LIN {X 0,Y 376.108,Z 924.328,A -85,B 0,C 180,E1 13646.479,E2 13646.479} C_VEL
LIN {X 0,Y 367.775,Z 908.146,A -85,B 0,C 180,E1 13649.429,E2 13649.429} C_VEL
LIN {X 0,Y 364.4,Z 915.516,A -85,B 0,C 180,E1 13649.758,E2 13649.758} C_VEL
LIN {X 0,Y 357.895,Z 928.85,A -85,B 0,C 180,E1 13650.369,E2 13650.369} C_VEL
LIN {X 0,Y 353.873,Z 934.95,A -85,B 0,C 180,E1 13650.878,E2 13650.878} C_VEL
LIN {X 0,Y 348.654,Z 943.219,A -85,B 0,C 180,E1 13651.467,E2 13651.467} C_VEL
LIN {X 0,Y 345.906,Z 946.107,A -85,B 0,C 180,E1 13652.021,E2 13652.021} C_VEL
LIN {X 0,Y 343.36,Z 977.029,A -85,B 0,C 180,E1 13654.434,E2 13654.434} C_VEL
LIN {X 0,Y 340.02,Z 1003.082,A -85,B 0,C 180,E1 13657.588,E2 13657.588} C_VEL
LIN {X 0,Y 336.523,Z 1024.234,A -85,B 0,C 180,E1 13661.411,E2 13661.411} C_VEL
LIN {X 0,Y 333.51,Z 1039.452,A -85,B 0,C 180,E1 13665.541,E2 13665.541} C_VEL
LIN {X 0,Y 331.006,Z 1050.175,A -85,B 0,C 180,E1 13670.2,E2 13670.2} C_VEL
LIN {X 0,Y 329.716,Z 1055.388,A -85,B 0,C 180,E1 13674.73,E2 13674.73} C_VEL
LIN {X 0,Y 328.873,Z 1055.973,A -85,B 0,C 180,E1 13679.999,E2 13679.999} C_VEL
LIN {X 0,Y 328.837,Z 1050.81,A -85,B 0,C 180,E1 13685.282,E2 13685.282} C_VEL
LIN {X 0,Y 329.705,Z 1039.548,A -85,B 0,C 180,E1 13690.582,E2 13690.582} C_VEL
LIN {X 0,Y 331.439,Z 1023.575,A -85,B 0,C 180,E1 13695.226,E2 13695.226} C_VEL
LIN {X 0,Y 334.022,Z 1001.735,A -85,B 0,C 180,E1 13699.527,E2 13699.527} C_VEL
LIN {X 0,Y 337.182,Z 974.565,A -85,B 0,C 180,E1 13703.187,E2 13703.187} C_VEL
LIN {X 0,Y 339.904,Z 944.159,A -85,B 0,C 180,E1 13705.915,E2 13705.915} C_VEL
LIN {X 0,Y 341.977,Z 913.832,A -85,B 0,C 180,E1 13707.697,E2 13707.697} C_VEL
LIN {X 0,Y 345.152,Z 909.514,A -85,B 0,C 180,E1 13708.423,E2 13708.423} C_VEL
LIN {X 0,Y 349.954,Z 896.791,A -85,B 0,C 180,E1 13709.156,E2 13709.156} C_VEL
LIN {X 0,Y 354.172,Z 888.97,A -85,B 0,C 180,E1 13710.083,E2 13710.083} C_VEL
LIN {X 0,Y 355.518,Z 886.512,A -85,B 0,C 180,E1 13710.372,E2 13710.372} C_VEL
LIN {X 0,Y 370.198,Z 910.648,A -85,B 0,C 180,E1 13715.495,E2 13715.495} C_VEL
LIN {X 0,Y 383.568,Z 939.518,A -85,B 0,C 180,E1 13720.262,E2 13720.262} C_VEL
LIN {X 0,Y 386.458,Z 948.208,A -85,B 0,C 180,E1 13721.491,E2 13721.491} C_VEL
LIN {X 0,Y 378.77,Z 984.053,A -85,B 0,C 180,E1 13723.63,E2 13723.63} C_VEL
LIN {X 0,Y 369.066,Z 1018.522,A -85,B 0,C 180,E1 13726.591,E2 13726.591} C_VEL
LIN {X 0,Y 358.745,Z 1049.661,A -85,B 0,C 180,E1 13730.368,E2 13730.368} C_VEL
LIN {X 0,Y 348.828,Z 1076.763,A -85,B 0,C 180,E1 13734.89,E2 13734.89} C_VEL
LIN {X 0,Y 339.261,Z 1101.55,A -85,B 0,C 180,E1 13740.597,E2 13740.597} C_VEL
LIN {X 0,Y 332.687,Z 1119.974,A -85,B 0,C 180,E1 13746.531,E2 13746.531} C_VEL
LIN {X 0,Y 328.362,Z 1134.473,A -85,B 0,C 180,E1 13753.249,E2 13753.249} C_VEL
LIN {X 0,Y 326.282,Z 1144.274,A -85,B 0,C 180,E1 13760.651,E2 13760.651} C_VEL
LIN {X 0,Y 325.694,Z 1148.277,A -85,B 0,C 180,E1 13767.334,E2 13767.334} C_VEL
LIN {X 0,Y 325.744,Z 1148.241,A -85,B 0,C 180,E1 13772.663,E2 13772.663} C_VEL
LIN {X 0,Y 326.287,Z 1144.195,A -85,B 0,C 180,E1 13779.346,E2 13779.346} C_VEL
LIN {X 0,Y 328.377,Z 1134.321,A -85,B 0,C 180,E1 13786.748,E2 13786.748} C_VEL
LIN {X 0,Y 332.774,Z 1119.754,A -85,B 0,C 180,E1 13793.46,E2 13793.46} C_VEL
LIN {X 0,Y 340.29,Z 1099.046,A -85,B 0,C 180,E1 13799.987,E2 13799.987} C_VEL
LIN {X 0,Y 350.198,Z 1073.11,A -85,B 0,C 180,E1 13805.709,E2 13805.709} C_VEL
LIN {X 0,Y 360.949,Z 1043.194,A -85,B 0,C 180,E1 13810.431,E2 13810.431} C_VEL
LIN {X 0,Y 371.664,Z 1010.049,A -85,B 0,C 180,E1 13814.133,E2 13814.133} C_VEL
LIN {X 0,Y 381.081,Z 973.71,A -85,B 0,C 180,E1 13816.999,E2 13816.999} C_VEL
LIN {X 0,Y 386.353,Z 946.977,A -85,B 0,C 180,E1 13818.517,E2 13818.517} C_VEL
LIN {X 0,Y 374.373,Z 918.78,A -85,B 0,C 180,E1 13822.931,E2 13822.931} C_VEL
LIN {X 0,Y 360.213,Z 893.932,A -85,B 0,C 180,E1 13827.801,E2 13827.801} C_VEL
LIN {X 0,Y 347.294,Z 875.046,A -85,B 0,C 180,E1 13832.671,E2 13832.671} C_VEL
LIN {X 0,Y 339.642,Z 864.701,A -85,B 0,C 180,E1 13836.146,E2 13836.146} C_VEL
LIN {X 0,Y 334.753,Z 857.931,A -85,B 0,C 180,E1 13838.79,E2 13838.79} C_VEL
LIN {X 0,Y 330.751,Z 852.629,A -85,B 0,C 180,E1 13841.314,E2 13841.314} C_VEL
LIN {X 0,Y 329.425,Z 850.767,A -85,B 0,C 180,E1 13842.257,E2 13842.257} C_VEL
LIN {X 0,Y 325.061,Z 845.874,A -85,B 0,C 180,E1 13845.848,E2 13845.848} C_VEL
LIN {X 0,Y 324.743,Z 843.44,A -85,B 0,C 180,E1 13846.522,E2 13846.522} C_VEL
LIN {X 0,Y 325.226,Z 843.44,A -85,B 0,C 180,E1 13854.659,E2 13854.659} C_VEL
LIN {X 0,Y 325.59,Z 843.44,A -85,B 0,C 180,E1 13860.001,E2 13860.001} C_VEL
LIN {X 0,Y 324.995,Z 843.44,A -85,B 0,C 180,E1 13868.035,E2 13868.035} C_VEL
LIN {X 0,Y 324.861,Z 844.009,A -85,B 0,C 180,E1 13869.304,E2 13869.304} C_VEL
LIN {X 0,Y 327.183,Z 849.216,A -85,B 0,C 180,E1 13871.617,E2 13871.617} C_VEL
LIN {X 0,Y 330.663,Z 851.939,A -85,B 0,C 180,E1 13874.079,E2 13874.079} C_VEL
LIN {X 0,Y 334.613,Z 857.811,A -85,B 0,C 180,E1 13876.641,E2 13876.641} C_VEL
LIN {X 0,Y 336.707,Z 860.625,A -85,B 0,C 180,E1 13877.835,E2 13877.835} C_VEL
LIN {X 0,Y 342.23,Z 868.171,A -85,B 0,C 180,E1 13880.646,E2 13880.646} C_VEL
LIN {X 0,Y 351.334,Z 880.835,A -85,B 0,C 180,E1 13884.527,E2 13884.527} C_VEL
LIN {X 0,Y 365.006,Z 902.571,A -85,B 0,C 180,E1 13889.594,E2 13889.594} C_VEL
LIN {X 0,Y 378.204,Z 929.229,A -85,B 0,C 180,E1 13894.346,E2 13894.346} C_VEL
LIN {X 0,Y 385.902,Z 951.03,A -85,B 0,C 180,E1 13897.51,E2 13897.51} C_VEL
LIN {X 0,Y 376.987,Z 993.57,A -85,B 0,C 180,E1 13900.262,E2 13900.262} C_VEL
LIN {X 0,Y 366.594,Z 1031.143,A -85,B 0,C 180,E1 13903.716,E2 13903.716} C_VEL
LIN {X 0,Y 355.486,Z 1065.912,A -85,B 0,C 180,E1 13908.156,E2 13908.156} C_VEL
LIN {X 0,Y 344.895,Z 1097.163,A -85,B 0,C 180,E1 13913.655,E2 13913.655} C_VEL
LIN {X 0,Y 336.481,Z 1122.605,A -85,B 0,C 180,E1 13919.764,E2 13919.764} C_VEL
LIN {X 0,Y 330.265,Z 1143.966,A -85,B 0,C 180,E1 13926.842,E2 13926.842} C_VEL
LIN {X 0,Y 327.114,Z 1158.659,A -85,B 0,C 180,E1 13933.877,E2 13933.877} C_VEL
LIN {X 0,Y 325.913,Z 1167.658,A -85,B 0,C 180,E1 13940.643,E2 13940.643} C_VEL
LIN {X 0,Y 325.706,Z 1171.943,A -85,B 0,C 180,E1 13947.337,E2 13947.337} C_VEL
LIN {X 0,Y 325.641,Z 1171.94,A -85,B 0,C 180,E1 13952.666,E2 13952.666} C_VEL
LIN {X 0,Y 325.91,Z 1167.658,A -85,B 0,C 180,E1 13959.359,E2 13959.359} C_VEL
LIN {X 0,Y 327.121,Z 1158.659,A -85,B 0,C 180,E1 13966.125,E2 13966.125} C_VEL
LIN {X 0,Y 330.278,Z 1143.971,A -85,B 0,C 180,E1 13973.159,E2 13973.159} C_VEL
LIN {X 0,Y 336.415,Z 1122.636,A -85,B 0,C 180,E1 13980.237,E2 13980.237} C_VEL
LIN {X 0,Y 338.564,Z 1116.059,A -85,B 0,C 180,E1 13981.992,E2 13981.992} C_VEL
LIN {X 0,Y 338.171,Z 1107.045,A -85,B 0,C 180,E1 13984.532,E2 13984.532} C_VEL
LIN {X 0,Y 338.05,Z 1097.476,A -85,B 0,C 180,E1 13987.029,E2 13987.029} C_VEL
LIN {X 0,Y 349.215,Z 1066.113,A -85,B 0,C 180,E1 13992.655,E2 13992.655} C_VEL
LIN {X 0,Y 361.147,Z 1029.977,A -85,B 0,C 180,E1 13997.312,E2 13997.312} C_VEL
LIN {X 0,Y 372.132,Z 991.554,A -85,B 0,C 180,E1 14000.812,E2 14000.812} C_VEL
LIN {X 0,Y 380.39,Z 954.941,A -85,B 0,C 180,E1 14003.166,E2 14003.166} C_VEL
LIN {X 0,Y 371.021,Z 928.372,A -85,B 0,C 180,E1 14007.27,E2 14007.27} C_VEL
LIN {X 0,Y 366.968,Z 920.536,A -85,B 0,C 180,E1 14008.782,E2 14008.782} C_VEL
LIN {X 0,Y 359.568,Z 934.219,A -85,B 0,C 180,E1 14009.476,E2 14009.476} C_VEL
LIN {X 0,Y 350.055,Z 948.399,A -85,B 0,C 180,E1 14010.519,E2 14010.519} C_VEL
LIN {X 0,Y 340.44,Z 959.968,A -85,B 0,C 180,E1 14011.802,E2 14011.802} C_VEL
LIN {X 0,Y 338.533,Z 961.854,A -85,B 0,C 180,E1 14012.264,E2 14012.264} C_VEL
LIN {X 0,Y 335.38,Z 990.271,A -85,B 0,C 180,E1 14015.018,E2 14015.018} C_VEL
LIN {X 0,Y 331.905,Z 1012.677,A -85,B 0,C 180,E1 14018.245,E2 14018.245} C_VEL
LIN {X 0,Y 328.372,Z 1031.449,A -85,B 0,C 180,E1 14022.214,E2 14022.214} C_VEL
LIN {X 0,Y 325.27,Z 1045.038,A -85,B 0,C 180,E1 14026.541,E2 14026.541} C_VEL
LIN {X 0,Y 323.081,Z 1053.423,A -85,B 0,C 180,E1 14030.93,E2 14030.93} C_VEL
LIN {X 0,Y 322.031,Z 1057.041,A -85,B 0,C 180,E1 14034.604,E2 14034.604} C_VEL
LIN {X 0,Y 321.112,Z 1057.42,A -85,B 0,C 180,E1 14039.999,E2 14039.999} C_VEL
LIN {X 0,Y 321.084,Z 1052.008,A -85,B 0,C 180,E1 14045.41,E2 14045.41} C_VEL
LIN {X 0,Y 321.743,Z 1042.227,A -85,B 0,C 180,E1 14050.161,E2 14050.161} C_VEL
LIN {X 0,Y 323.495,Z 1026.843,A -85,B 0,C 180,E1 14054.914,E2 14054.914} C_VEL
LIN {X 0,Y 326.047,Z 1005.884,A -85,B 0,C 180,E1 14059.318,E2 14059.318} C_VEL
LIN {X 0,Y 329.216,Z 979.656,A -85,B 0,C 180,E1 14063.094,E2 14063.094} C_VEL
LIN {X 0,Y 332.106,Z 949.359,A -85,B 0,C 180,E1 14066.024,E2 14066.024} C_VEL
LIN {X 0,Y 333.389,Z 936.954,A -85,B 0,C 180,E1 14067.006,E2 14067.006} C_VEL
LIN {X 0,Y 337.196,Z 932.766,A -85,B 0,C 180,E1 14067.905,E2 14067.905} C_VEL
LIN {X 0,Y 344.097,Z 918.915,A -85,B 0,C 180,E1 14068.872,E2 14068.872} C_VEL
LIN {X 0,Y 349.104,Z 909.69,A -85,B 0,C 180,E1 14069.726,E2 14069.726} C_VEL
LIN {X 0,Y 352.399,Z 901.513,A -85,B 0,C 180,E1 14070.21,E2 14070.21} C_VEL
LIN {X 0,Y 355.375,Z 897.164,A -85,B 0,C 180,E1 14070.839,E2 14070.839} C_VEL
LIN {X 0,Y 369.602,Z 923.178,A -85,B 0,C 180,E1 14076.163,E2 14076.163} C_VEL
LIN {X 0,Y 380.719,Z 949.941,A -85,B 0,C 180,E1 14080.564,E2 14080.564} C_VEL
LIN {X 0,Y 372.121,Z 989.556,A -85,B 0,C 180,E1 14083.105,E2 14083.105} C_VEL
LIN {X 0,Y 361.673,Z 1024.445,A -85,B 0,C 180,E1 14086.308,E2 14086.308} C_VEL
LIN {X 0,Y 349.978,Z 1057.121,A -85,B 0,C 180,E1 14090.582,E2 14090.582} C_VEL
LIN {X 0,Y 339.324,Z 1084.484,A -85,B 0,C 180,E1 14095.629,E2 14095.629} C_VEL
LIN {X 0,Y 330.036,Z 1107.705,A -85,B 0,C 180,E1 14101.615,E2 14101.615} C_VEL
LIN {X 0,Y 323.268,Z 1126.436,A -85,B 0,C 180,E1 14108.571,E2 14108.571} C_VEL
LIN {X 0,Y 319.816,Z 1138.047,A -85,B 0,C 180,E1 14114.905,E2 14114.905} C_VEL
LIN {X 0,Y 318.195,Z 1145.708,A -85,B 0,C 180,E1 14121.791,E2 14121.791} C_VEL
LIN {X 0,Y 317.815,Z 1148.564,A -85,B 0,C 180,E1 14127.268,E2 14127.268} C_VEL
LIN {X 0,Y 317.845,Z 1148.53,A -85,B 0,C 180,E1 14132.729,E2 14132.729} C_VEL
LIN {X 0,Y 318.441,Z 1144.488,A -85,B 0,C 180,E1 14139.578,E2 14139.578} C_VEL
LIN {X 0,Y 320.716,Z 1134.625,A -85,B 0,C 180,E1 14147.16,E2 14147.16} C_VEL
LIN {X 0,Y 325.391,Z 1120.071,A -85,B 0,C 180,E1 14154.025,E2 14154.025} C_VEL
LIN {X 0,Y 333.42,Z 1099.224,A -85,B 0,C 180,E1 14160.72,E2 14160.72} C_VEL
LIN {X 0,Y 343.708,Z 1073.49,A -85,B 0,C 180,E1 14166.491,E2 14166.491} C_VEL
LIN {X 0,Y 354.512,Z 1044.754,A -85,B 0,C 180,E1 14171.121,E2 14171.121} C_VEL
LIN {X 0,Y 365.807,Z 1011.321,A -85,B 0,C 180,E1 14174.927,E2 14174.927} C_VEL
LIN {X 0,Y 375.514,Z 975.542,A -85,B 0,C 180,E1 14177.803,E2 14177.803} C_VEL
LIN {X 0,Y 380.906,Z 950.822,A -85,B 0,C 180,E1 14179.22,E2 14179.22} C_VEL
LIN {X 0,Y 369.756,Z 923.356,A -85,B 0,C 180,E1 14183.673,E2 14183.673} C_VEL
LIN {X 0,Y 355.266,Z 897.107,A -85,B 0,C 180,E1 14189.064,E2 14189.064} C_VEL
LIN {X 0,Y 342.486,Z 878.43,A -85,B 0,C 180,E1 14194.279,E2 14194.279} C_VEL
LIN {X 0,Y 336.753,Z 870.971,A -85,B 0,C 180,E1 14197.062,E2 14197.062} C_VEL
LIN {X 0,Y 332.73,Z 865.184,A -85,B 0,C 180,E1 14199.353,E2 14199.353} C_VEL
LIN {X 0,Y 328.809,Z 859.258,A -85,B 0,C 180,E1 14201.981,E2 14201.981} C_VEL
LIN {X 0,Y 323.61,Z 853.281,A -85,B 0,C 180,E1 14206.301,E2 14206.301} C_VEL
LIN {X 0,Y 322.769,Z 851.097,A -85,B 0,C 180,E1 14207.316,E2 14207.316} C_VEL
LIN {X 0,Y 318.051,Z 846.227,A -85,B 0,C 180,E1 14218.639,E2 14218.639} C_VEL
LIN {X 0,Y 323.423,Z 851.958,A -85,B 0,C 180,E1 14228.921,E2 14228.921} C_VEL
LIN {X 0,Y 326.674,Z 857.585,A -85,B 0,C 180,E1 14232.012,E2 14232.012} C_VEL
LIN {X 0,Y 329.121,Z 859.853,A -85,B 0,C 180,E1 14233.775,E2 14233.775} C_VEL
LIN {X 0,Y 333.649,Z 865.777,A -85,B 0,C 180,E1 14236.69,E2 14236.69} C_VEL
LIN {X 0,Y 344.313,Z 881.028,A -85,B 0,C 180,E1 14242.118,E2 14242.118} C_VEL
LIN {X 0,Y 356.7,Z 900.459,A -85,B 0,C 180,E1 14247.237,E2 14247.237} C_VEL
LIN {X 0,Y 369.956,Z 925.813,A -85,B 0,C 180,E1 14252.314,E2 14252.314} C_VEL
LIN {X 0,Y 379.853,Z 952.241,A -85,B 0,C 180,E1 14256.501,E2 14256.501} C_VEL
LIN {X 0,Y 380.069,Z 956.725,A -85,B 0,C 180,E1 14256.958,E2 14256.958} C_VEL
LIN {X 0,Y 370.784,Z 996.439,A -85,B 0,C 180,E1 14259.578,E2 14259.578} C_VEL
LIN {X 0,Y 360.364,Z 1032.559,A -85,B 0,C 180,E1 14262.991,E2 14262.991} C_VEL
LIN {X 0,Y 348.9,Z 1066.802,A -85,B 0,C 180,E1 14267.455,E2 14267.455} C_VEL
LIN {X 0,Y 337.677,Z 1098.296,A -85,B 0,C 180,E1 14273.151,E2 14273.151} C_VEL
LIN {X 0,Y 328.734,Z 1124.026,A -85,B 0,C 180,E1 14279.56,E2 14279.56} C_VEL
LIN {X 0,Y 322.649,Z 1143.973,A -85,B 0,C 180,E1 14286.406,E2 14286.406} C_VEL
LIN {X 0,Y 319.329,Z 1158.344,A -85,B 0,C 180,E1 14293.473,E2 14293.473} C_VEL
LIN {X 0,Y 318.02,Z 1167.36,A -85,B 0,C 180,E1 14300.409,E2 14300.409} C_VEL
LIN {X 0,Y 317.824,Z 1171.655,A -85,B 0,C 180,E1 14307.271,E2 14307.271} C_VEL
LIN {X 0,Y 317.735,Z 1171.652,A -85,B 0,C 180,E1 14312.733,E2 14312.733} C_VEL
LIN {X 0,Y 318.019,Z 1167.361,A -85,B 0,C 180,E1 14319.594,E2 14319.594} C_VEL
LIN {X 0,Y 319.332,Z 1158.346,A -85,B 0,C 180,E1 14326.53,E2 14326.53} C_VEL
LIN {X 0,Y 322.996,Z 1142.722,A -85,B 0,C 180,E1 14334.083,E2 14334.083} C_VEL
LIN {X 0,Y 329.264,Z 1122.46,A -85,B 0,C 180,E1 14340.909,E2 14340.909} C_VEL
LIN {X 0,Y 338.05,Z 1097.476,A -85,B 0,C 180,E1 14347.029,E2 14347.029} C_VEL
LIN {X 0,Y 338.415,Z 1087.431,A -85,B 0,C 180,E1 14349.466,E2 14349.466} C_VEL
LIN {X 0,Y 339.081,Z 1076.685,A -85,B 0,C 180,E1 14351.808,E2 14351.808} C_VEL
LIN {X 0,Y 351.505,Z 1041.807,A -85,B 0,C 180,E1 14356.872,E2 14356.872} C_VEL
LIN {X 0,Y 363.28,Z 1004.627,A -85,B 0,C 180,E1 14360.687,E2 14360.687} C_VEL
LIN {X 0,Y 373.629,Z 964.087,A -85,B 0,C 180,E1 14363.575,E2 14363.575} C_VEL
LIN {X 0,Y 374.496,Z 956.807,A -85,B 0,C 180,E1 14364.111,E2 14364.111} C_VEL
LIN {X 0,Y 366.129,Z 932.669,A -85,B 0,C 180,E1 14368.033,E2 14368.033} C_VEL
LIN {X 0,Y 357.489,Z 945.376,A -85,B 0,C 180,E1 14368.932,E2 14368.932} C_VEL
LIN {X 0,Y 343.084,Z 963.636,A -85,B 0,C 180,E1 14370.578,E2 14370.578} C_VEL
LIN {X 0,Y 332.367,Z 974.04,A -85,B 0,C 180,E1 14372.166,E2 14372.166} C_VEL
LIN {X 0,Y 330.964,Z 976.184,A -85,B 0,C 180,E1 14372.593,E2 14372.593} C_VEL
LIN {X 0,Y 327.158,Z 1002.804,A -85,B 0,C 180,E1 14375.75,E2 14375.75} C_VEL
LIN {X 0,Y 323.078,Z 1024.626,A -85,B 0,C 180,E1 14379.609,E2 14379.609} C_VEL
LIN {X 0,Y 319.258,Z 1041.566,A -85,B 0,C 180,E1 14384.176,E2 14384.176} C_VEL
LIN {X 0,Y 316.253,Z 1052.612,A -85,B 0,C 180,E1 14388.959,E2 14388.959} C_VEL
LIN {X 0,Y 314.733,Z 1057.76,A -85,B 0,C 180,E1 14393.092,E2 14393.092} C_VEL
LIN {X 0,Y 313.707,Z 1059.518,A -85,B 0,C 180,E1 14397.233,E2 14397.233} C_VEL
LIN {X 0,Y 313.188,Z 1056.766,A -85,B 0,C 180,E1 14402.769,E2 14402.769} C_VEL
LIN {X 0,Y 313.606,Z 1048.112,A -85,B 0,C 180,E1 14408.326,E2 14408.326} C_VEL
LIN {X 0,Y 315.116,Z 1033.768,A -85,B 0,C 180,E1 14413.544,E2 14413.544} C_VEL
LIN {X 0,Y 317.612,Z 1013.374,A -85,B 0,C 180,E1 14418.411,E2 14418.411} C_VEL
LIN {X 0,Y 320.776,Z 988.318,A -85,B 0,C 180,E1 14422.493,E2 14422.493} C_VEL
LIN {X 0,Y 324.008,Z 958.281,A -85,B 0,C 180,E1 14425.792,E2 14425.792} C_VEL
LIN {X 0,Y 324.813,Z 954.885,A -85,B 0,C 180,E1 14426.281,E2 14426.281} C_VEL
LIN {X 0,Y 328.099,Z 952.113,A -85,B 0,C 180,E1 14427.106,E2 14427.106} C_VEL
LIN {X 0,Y 334.082,Z 943.064,A -85,B 0,C 180,E1 14428.043,E2 14428.043} C_VEL
LIN {X 0,Y 340.38,Z 934.73,A -85,B 0,C 180,E1 14429.199,E2 14429.199} C_VEL
LIN {X 0,Y 346.421,Z 923.149,A -85,B 0,C 180,E1 14429.98,E2 14429.98} C_VEL
LIN {X 0,Y 352.739,Z 910.791,A -85,B 0,C 180,E1 14430.909,E2 14430.909} C_VEL
LIN {X 0,Y 354.291,Z 907.223,A -85,B 0,C 180,E1 14431.14,E2 14431.14} C_VEL
LIN {X 0,Y 366.853,Z 932.075,A -85,B 0,C 180,E1 14436.202,E2 14436.202} C_VEL
LIN {X 0,Y 375.175,Z 954.807,A -85,B 0,C 180,E1 14439.931,E2 14439.931} C_VEL
LIN {X 0,Y 365.799,Z 993.304,A -85,B 0,C 180,E1 14442.453,E2 14442.453} C_VEL
LIN {X 0,Y 355.069,Z 1027.381,A -85,B 0,C 180,E1 14445.709,E2 14445.709} C_VEL
LIN {X 0,Y 343.504,Z 1058.272,A -85,B 0,C 180,E1 14449.859,E2 14449.859} C_VEL
LIN {X 0,Y 332.198,Z 1086.004,A -85,B 0,C 180,E1 14455.115,E2 14455.115} C_VEL
LIN {X 0,Y 322.436,Z 1109.231,A -85,B 0,C 180,E1 14461.325,E2 14461.325} C_VEL
LIN {X 0,Y 315.43,Z 1127.654,A -85,B 0,C 180,E1 14468.471,E2 14468.471} C_VEL
LIN {X 0,Y 311.605,Z 1140.214,A -85,B 0,C 180,E1 14475.938,E2 14475.938} C_VEL
LIN {X 0,Y 310.33,Z 1146,A -85,B 0,C 180,E1 14481.582,E2 14481.582} C_VEL
LIN {X 0,Y 309.913,Z 1148.852,A -85,B 0,C 180,E1 14487.198,E2 14487.198} C_VEL
LIN {X 0,Y 309.942,Z 1148.818,A -85,B 0,C 180,E1 14492.799,E2 14492.799} C_VEL
LIN {X 0,Y 310.594,Z 1144.78,A -85,B 0,C 180,E1 14499.823,E2 14499.823} C_VEL
LIN {X 0,Y 313.05,Z 1134.928,A -85,B 0,C 180,E1 14507.594,E2 14507.594} C_VEL
LIN {X 0,Y 318.024,Z 1120.387,A -85,B 0,C 180,E1 14514.618,E2 14514.618} C_VEL
LIN {X 0,Y 326.514,Z 1099.562,A -85,B 0,C 180,E1 14521.444,E2 14521.444} C_VEL
LIN {X 0,Y 337.279,Z 1073.868,A -85,B 0,C 180,E1 14527.303,E2 14527.303} C_VEL
LIN {X 0,Y 348.828,Z 1044.38,A -85,B 0,C 180,E1 14532.09,E2 14532.09} C_VEL
LIN {X 0,Y 360.679,Z 1010.351,A -85,B 0,C 180,E1 14535.959,E2 14535.959} C_VEL
LIN {X 0,Y 370.559,Z 975.031,A -85,B 0,C 180,E1 14538.781,E2 14538.781} C_VEL
LIN {X 0,Y 375.158,Z 953.689,A -85,B 0,C 180,E1 14540.069,E2 14540.069} C_VEL
LIN {X 0,Y 364.571,Z 926.844,A -85,B 0,C 180,E1 14544.637,E2 14544.637} C_VEL
LIN {X 0,Y 351.223,Z 902.282,A -85,B 0,C 180,E1 14549.964,E2 14549.964} C_VEL
LIN {X 0,Y 340.245,Z 885.439,A -85,B 0,C 180,E1 14554.789,E2 14554.789} C_VEL
LIN {X 0,Y 331.019,Z 872.548,A -85,B 0,C 180,E1 14559.766,E2 14559.766} C_VEL
LIN {X 0,Y 325.976,Z 865.718,A -85,B 0,C 180,E1 14563.301,E2 14563.301} C_VEL
LIN {X 0,Y 321.999,Z 859.946,A -85,B 0,C 180,E1 14567.01,E2 14567.01} C_VEL
LIN {X 0,Y 317.952,Z 856.269,A -85,B 0,C 180,E1 14572.821,E2 14572.821} C_VEL
LIN {X 0,Y 317.067,Z 854.053,A -85,B 0,C 180,E1 14577.264,E2 14577.264} C_VEL
LIN {X 0,Y 318.058,Z 855.967,A -85,B 0,C 180,E1 14582.858,E2 14582.858} C_VEL
LIN {X 0,Y 322.111,Z 859.902,A -85,B 0,C 180,E1 14588.639,E2 14588.639} C_VEL
LIN {X 0,Y 325.867,Z 865.606,A -85,B 0,C 180,E1 14592.169,E2 14592.169} C_VEL
LIN {X 0,Y 327.856,Z 868.207,A -85,B 0,C 180,E1 14593.669,E2 14593.669} C_VEL
LIN {X 0,Y 333.357,Z 875.955,A -85,B 0,C 180,E1 14597.219,E2 14597.219} C_VEL
LIN {X 0,Y 341.741,Z 887.684,A -85,B 0,C 180,E1 14601.557,E2 14601.557} C_VEL
LIN {X 0,Y 354.19,Z 908.118,A -85,B 0,C 180,E1 14607.012,E2 14607.012} C_VEL
LIN {X 0,Y 366.285,Z 933.103,A -85,B 0,C 180,E1 14612.065,E2 14612.065} C_VEL
LIN {X 0,Y 374.524,Z 956.516,A -85,B 0,C 180,E1 14615.886,E2 14615.886} C_VEL
LIN {X 0,Y 372.959,Z 966.546,A -85,B 0,C 180,E1 14616.556,E2 14616.556} C_VEL
LIN {X 0,Y 362.235,Z 1007.794,A -85,B 0,C 180,E1 14619.587,E2 14619.587} C_VEL
LIN {X 0,Y 350.39,Z 1045.125,A -85,B 0,C 180,E1 14623.562,E2 14623.562} C_VEL
LIN {X 0,Y 338.827,Z 1077.336,A -85,B 0,C 180,E1 14628.313,E2 14628.313} C_VEL
LIN {X 0,Y 327.866,Z 1106.392,A -85,B 0,C 180,E1 14634.198,E2 14634.198} C_VEL
LIN {X 0,Y 319.16,Z 1130.952,A -85,B 0,C 180,E1 14641.103,E2 14641.103} C_VEL
LIN {X 0,Y 313.379,Z 1150.163,A -85,B 0,C 180,E1 14648.755,E2 14648.755} C_VEL
LIN {X 0,Y 310.81,Z 1162.263,A -85,B 0,C 180,E1 14655.903,E2 14655.903} C_VEL
LIN {X 0,Y 310.035,Z 1168.344,A -85,B 0,C 180,E1 14661.576,E2 14661.576} C_VEL
LIN {X 0,Y 309.915,Z 1171.366,A -85,B 0,C 180,E1 14667.201,E2 14667.201} C_VEL
LIN {X 0,Y 309.83,Z 1171.364,A -85,B 0,C 180,E1 14672.802,E2 14672.802} C_VEL
LIN {X 0,Y 310.132,Z 1167.065,A -85,B 0,C 180,E1 14679.84,E2 14679.84} C_VEL
LIN {X 0,Y 311.575,Z 1158.035,A -85,B 0,C 180,E1 14686.954,E2 14686.954} C_VEL
LIN {X 0,Y 315.059,Z 1143.928,A -85,B 0,C 180,E1 14694.074,E2 14694.074} C_VEL
LIN {X 0,Y 322.029,Z 1122.57,A -85,B 0,C 180,E1 14701.534,E2 14701.534} C_VEL
LIN {X 0,Y 331.701,Z 1096.434,A -85,B 0,C 180,E1 14708.044,E2 14708.044} C_VEL
LIN {X 0,Y 339.081,Z 1076.685,A -85,B 0,C 180,E1 14711.808,E2 14711.808} C_VEL
LIN {X 0,Y 340.227,Z 1065.527,A -85,B 0,C 180,E1 14714.088,E2 14714.088} C_VEL
LIN {X 0,Y 341.468,Z 1053.726,A -85,B 0,C 180,E1 14716.261,E2 14716.261} C_VEL
LIN {X 0,Y 354.179,Z 1016.874,A -85,B 0,C 180,E1 14720.533,E2 14720.533} C_VEL
LIN {X 0,Y 365.401,Z 977.956,A -85,B 0,C 180,E1 14723.673,E2 14723.673} C_VEL
LIN {X 0,Y 369.162,Z 960.803,A -85,B 0,C 180,E1 14724.78,E2 14724.78} C_VEL
LIN {X 0,Y 364.387,Z 945.395,A -85,B 0,C 180,E1 14727.307,E2 14727.307} C_VEL
LIN {X 0,Y 363.309,Z 944.323,A -85,B 0,C 180,E1 14727.654,E2 14727.654} C_VEL
LIN {X 0,Y 352.327,Z 959.303,A -85,B 0,C 180,E1 14728.703,E2 14728.703} C_VEL
LIN {X 0,Y 342.3,Z 970.563,A -85,B 0,C 180,E1 14729.854,E2 14729.854} C_VEL
LIN {X 0,Y 325.479,Z 985.846,A -85,B 0,C 180,E1 14732.279,E2 14732.279} C_VEL
LIN {X 0,Y 323.373,Z 987.722,A -85,B 0,C 180,E1 14732.831,E2 14732.831} C_VEL
LIN {X 0,Y 319.255,Z 1012.164,A -85,B 0,C 180,E1 14736.228,E2 14736.228} C_VEL
LIN {X 0,Y 314.94,Z 1032.109,A -85,B 0,C 180,E1 14740.335,E2 14740.335} C_VEL
LIN {X 0,Y 310.941,Z 1047.434,A -85,B 0,C 180,E1 14745.188,E2 14745.188} C_VEL
LIN {X 0,Y 308.19,Z 1056.264,A -85,B 0,C 180,E1 14749.835,E2 14749.835} C_VEL
LIN {X 0,Y 306.67,Z 1060.392,A -85,B 0,C 180,E1 14754.332,E2 14754.332} C_VEL
LIN {X 0,Y 305.604,Z 1060.3,A -85,B 0,C 180,E1 14759.999,E2 14759.999} C_VEL
LIN {X 0,Y 305.55,Z 1054.37,A -85,B 0,C 180,E1 14765.686,E2 14765.686} C_VEL
LIN {X 0,Y 306.284,Z 1044.024,A -85,B 0,C 180,E1 14770.681,E2 14770.681} C_VEL
LIN {X 0,Y 308.232,Z 1027.944,A -85,B 0,C 180,E1 14775.671,E2 14775.671} C_VEL
LIN {X 0,Y 310.998,Z 1005.965,A -85,B 0,C 180,E1 14780.293,E2 14780.293} C_VEL
LIN {X 0,Y 314.436,Z 979.278,A -85,B 0,C 180,E1 14784.133,E2 14784.133} C_VEL
LIN {X 0,Y 315.578,Z 969.989,A -85,B 0,C 180,E1 14785.242,E2 14785.242} C_VEL
LIN {X 0,Y 319.649,Z 967.13,A -85,B 0,C 180,E1 14786.361,E2 14786.361} C_VEL
LIN {X 0,Y 323.846,Z 961.769,A -85,B 0,C 180,E1 14787.041,E2 14787.041} C_VEL
LIN {X 0,Y 329.289,Z 956.585,A -85,B 0,C 180,E1 14788.228,E2 14788.228} C_VEL
LIN {X 0,Y 336.339,Z 947.117,A -85,B 0,C 180,E1 14789.333,E2 14789.333} C_VEL
LIN {X 0,Y 344.081,Z 935.819,A -85,B 0,C 180,E1 14790.487,E2 14790.487} C_VEL
LIN {X 0,Y 348.993,Z 926.904,A -85,B 0,C 180,E1 14791.096,E2 14791.096} C_VEL
LIN {X 0,Y 353.725,Z 918.905,A -85,B 0,C 180,E1 14791.815,E2 14791.815} C_VEL
LIN {X 0,Y 364.625,Z 942.99,A -85,B 0,C 180,E1 14796.613,E2 14796.613} C_VEL
LIN {X 0,Y 369.71,Z 957.835,A -85,B 0,C 180,E1 14799.126,E2 14799.126} C_VEL
LIN {X 0,Y 360.292,Z 994.552,A -85,B 0,C 180,E1 14801.581,E2 14801.581} C_VEL
LIN {X 0,Y 349.408,Z 1027.823,A -85,B 0,C 180,E1 14804.796,E2 14804.796} C_VEL
LIN {X 0,Y 337.173,Z 1059.212,A -85,B 0,C 180,E1 14809.073,E2 14809.073} C_VEL
LIN {X 0,Y 325.639,Z 1086.345,A -85,B 0,C 180,E1 14814.306,E2 14814.306} C_VEL
LIN {X 0,Y 315.84,Z 1108.327,A -85,B 0,C 180,E1 14820.205,E2 14820.205} C_VEL
LIN {X 0,Y 308.731,Z 1125.876,A -85,B 0,C 180,E1 14826.898,E2 14826.898} C_VEL
LIN {X 0,Y 304.336,Z 1138.648,A -85,B 0,C 180,E1 14834.118,E2 14834.118} C_VEL
LIN {X 0,Y 302.468,Z 1146.291,A -85,B 0,C 180,E1 14841.361,E2 14841.361} C_VEL
LIN {X 0,Y 302.012,Z 1149.14,A -85,B 0,C 180,E1 14847.125,E2 14847.125} C_VEL
LIN {X 0,Y 302.04,Z 1149.107,A -85,B 0,C 180,E1 14852.872,E2 14852.872} C_VEL
LIN {X 0,Y 302.74,Z 1145.073,A -85,B 0,C 180,E1 14860.08,E2 14860.08} C_VEL
LIN {X 0,Y 305.389,Z 1135.23,A -85,B 0,C 180,E1 14868.051,E2 14868.051} C_VEL
LIN {X 0,Y 311.452,Z 1118.902,A -85,B 0,C 180,E1 14875.945,E2 14875.945} C_VEL
LIN {X 0,Y 320.227,Z 1098.619,A -85,B 0,C 180,E1 14882.536,E2 14882.536} C_VEL
LIN {X 0,Y 331.61,Z 1072.534,A -85,B 0,C 180,E1 14888.469,E2 14888.469} C_VEL
LIN {X 0,Y 343.734,Z 1042.755,A -85,B 0,C 180,E1 14893.254,E2 14893.254} C_VEL
LIN {X 0,Y 355.616,Z 1009.639,A -85,B 0,C 180,E1 14896.99,E2 14896.99} C_VEL
LIN {X 0,Y 365.673,Z 974.72,A -85,B 0,C 180,E1 14899.771,E2 14899.771} C_VEL
LIN {X 0,Y 369.723,Z 957.465,A -85,B 0,C 180,E1 14900.794,E2 14900.794} C_VEL
LIN {X 0,Y 360.06,Z 931.876,A -85,B 0,C 180,E1 14905.325,E2 14905.325} C_VEL
LIN {X 0,Y 347.866,Z 908.339,A -85,B 0,C 180,E1 14910.616,E2 14910.616} C_VEL
LIN {X 0,Y 337.653,Z 891.982,A -85,B 0,C 180,E1 14915.431,E2 14915.431} C_VEL
LIN {X 0,Y 328.959,Z 879.649,A -85,B 0,C 180,E1 14920.4,E2 14920.4} C_VEL
LIN {X 0,Y 324.626,Z 873.357,A -85,B 0,C 180,E1 14923.578,E2 14923.578} C_VEL
LIN {X 0,Y 320.608,Z 867.287,A -85,B 0,C 180,E1 14927.473,E2 14927.473} C_VEL
LIN {X 0,Y 316.102,Z 861.921,A -85,B 0,C 180,E1 14937.256,E2 14937.256} C_VEL
LIN {X 0,Y 317.038,Z 863.785,A -85,B 0,C 180,E1 14942.738,E2 14942.738} C_VEL
LIN {X 0,Y 320.821,Z 867.736,A -85,B 0,C 180,E1 14948.353,E2 14948.353} C_VEL
LIN {X 0,Y 325.063,Z 873.619,A -85,B 0,C 180,E1 14952.326,E2 14952.326} C_VEL
LIN {X 0,Y 331.839,Z 883.849,A -85,B 0,C 180,E1 14957.013,E2 14957.013} C_VEL
LIN {X 0,Y 339.78,Z 895.429,A -85,B 0,C 180,E1 14961.289,E2 14961.289} C_VEL
LIN {X 0,Y 351.474,Z 915.704,A -85,B 0,C 180,E1 14966.805,E2 14966.805} C_VEL
LIN {X 0,Y 362.469,Z 940.191,A -85,B 0,C 180,E1 14971.783,E2 14971.783} C_VEL
LIN {X 0,Y 369.18,Z 960.533,A -85,B 0,C 180,E1 14975.218,E2 14975.218} C_VEL
LIN {X 0,Y 359.248,Z 999.984,A -85,B 0,C 180,E1 14977.97,E2 14977.97} C_VEL
LIN {X 0,Y 348.414,Z 1034.293,A -85,B 0,C 180,E1 14981.33,E2 14981.33} C_VEL
LIN {X 0,Y 336.454,Z 1067.146,A -85,B 0,C 180,E1 14985.745,E2 14985.745} C_VEL
LIN {X 0,Y 324.597,Z 1097.557,A -85,B 0,C 180,E1 14991.4,E2 14991.4} C_VEL
LIN {X 0,Y 314.586,Z 1123.339,A -85,B 0,C 180,E1 14998.034,E2 14998.034} C_VEL
LIN {X 0,Y 307.588,Z 1143.599,A -85,B 0,C 180,E1 15005.305,E2 15005.305} C_VEL
LIN {X 0,Y 303.577,Z 1158.907,A -85,B 0,C 180,E1 15013.336,E2 15013.336} C_VEL
LIN {X 0,Y 302.257,Z 1166.767,A -85,B 0,C 180,E1 15019.903,E2 15019.903} C_VEL
LIN {X 0,Y 302.008,Z 1171.078,A -85,B 0,C 180,E1 15027.128,E2 15027.128} C_VEL
LIN {X 0,Y 301.941,Z 1171.076,A -85,B 0,C 180,E1 15032.876,E2 15032.876} C_VEL
LIN {X 0,Y 302.257,Z 1166.77,A -85,B 0,C 180,E1 15040.099,E2 15040.099} C_VEL
LIN {X 0,Y 303.805,Z 1157.726,A -85,B 0,C 180,E1 15047.401,E2 15047.401} C_VEL
LIN {X 0,Y 307.576,Z 1143.609,A -85,B 0,C 180,E1 15054.698,E2 15054.698} C_VEL
LIN {X 0,Y 314.993,Z 1122.225,A -85,B 0,C 180,E1 15062.323,E2 15062.323} C_VEL
LIN {X 0,Y 325.239,Z 1096.063,A -85,B 0,C 180,E1 15068.94,E2 15068.94} C_VEL
LIN {X 0,Y 337.548,Z 1064.435,A -85,B 0,C 180,E1 15074.685,E2 15074.685} C_VEL
LIN {X 0,Y 341.468,Z 1053.726,A -85,B 0,C 180,E1 15076.261,E2 15076.261} C_VEL
LIN {X 0,Y 342.999,Z 1041.438,A -85,B 0,C 180,E1 15078.354,E2 15078.354} C_VEL
LIN {X 0,Y 344.387,Z 1030.372,A -85,B 0,C 180,E1 15080.102,E2 15080.102} C_VEL
LIN {X 0,Y 344.947,Z 1028.598,A -85,B 0,C 180,E1 15080.297,E2 15080.297} C_VEL
LIN {X 0,Y 356.822,Z 991.17,A -85,B 0,C 180,E1 15083.732,E2 15083.732} C_VEL
LIN {X 0,Y 363.597,Z 963.888,A -85,B 0,C 180,E1 15085.622,E2 15085.622} C_VEL
LIN {X 0,Y 360.795,Z 956.005,A -85,B 0,C 180,E1 15087.072,E2 15087.072} C_VEL
LIN {X 0,Y 343.119,Z 975.972,A -85,B 0,C 180,E1 15088.9,E2 15088.9} C_VEL
LIN {X 0,Y 324.64,Z 992.101,A -85,B 0,C 180,E1 15091.443,E2 15091.443} C_VEL
LIN {X 0,Y 315.702,Z 998.722,A -85,B 0,C 180,E1 15093.159,E2 15093.159} C_VEL
LIN {X 0,Y 310.808,Z 1022.469,A -85,B 0,C 180,E1 15097.064,E2 15097.064} C_VEL
LIN {X 0,Y 306.297,Z 1040.769,A -85,B 0,C 180,E1 15101.632,E2 15101.632} C_VEL
LIN {X 0,Y 302.643,Z 1052.705,A -85,B 0,C 180,E1 15106.253,E2 15106.253} C_VEL
LIN {X 0,Y 300.044,Z 1060.05,A -85,B 0,C 180,E1 15111.292,E2 15111.292} C_VEL
LIN {X 0,Y 298.275,Z 1062.65,A -85,B 0,C 180,E1 15117.089,E2 15117.089} C_VEL
LIN {X 0,Y 297.641,Z 1059.372,A -85,B 0,C 180,E1 15122.914,E2 15122.914} C_VEL
LIN {X 0,Y 297.989,Z 1051.383,A -85,B 0,C 180,E1 15128.119,E2 15128.119} C_VEL
LIN {X 0,Y 299.465,Z 1037.443,A -85,B 0,C 180,E1 15133.52,E2 15133.52} C_VEL
LIN {X 0,Y 302.074,Z 1017.253,A -85,B 0,C 180,E1 15138.631,E2 15138.631} C_VEL
LIN {X 0,Y 305.405,Z 992.176,A -85,B 0,C 180,E1 15142.976,E2 15142.976} C_VEL
LIN {X 0,Y 306.561,Z 983.177,A -85,B 0,C 180,E1 15144.183,E2 15144.183} C_VEL
LIN {X 0,Y 310.754,Z 980.687,A -85,B 0,C 180,E1 15145.459,E2 15145.459} C_VEL
LIN {X 0,Y 315.801,Z 975.8,A -85,B 0,C 180,E1 15146.5,E2 15146.5} C_VEL
LIN {X 0,Y 321.851,Z 970.141,A -85,B 0,C 180,E1 15147.765,E2 15147.765} C_VEL
LIN {X 0,Y 332.735,Z 958.262,A -85,B 0,C 180,E1 15149.656,E2 15149.656} C_VEL
LIN {X 0,Y 345.032,Z 941.881,A -85,B 0,C 180,E1 15151.424,E2 15151.424} C_VEL
LIN {X 0,Y 351.985,Z 929.981,A -85,B 0,C 180,E1 15152.248,E2 15152.248} C_VEL
LIN {X 0,Y 359.554,Z 947.067,A -85,B 0,C 180,E1 15155.813,E2 15155.813} C_VEL
LIN {X 0,Y 364.145,Z 961.523,A -85,B 0,C 180,E1 15158.33,E2 15158.33} C_VEL
LIN {X 0,Y 353.668,Z 999.781,A -85,B 0,C 180,E1 15161.011,E2 15161.011} C_VEL
LIN {X 0,Y 341.547,Z 1034.459,A -85,B 0,C 180,E1 15164.594,E2 15164.594} C_VEL
LIN {X 0,Y 328.275,Z 1066.487,A -85,B 0,C 180,E1 15169.344,E2 15169.344} C_VEL
LIN {X 0,Y 315.692,Z 1094.138,A -85,B 0,C 180,E1 15175.279,E2 15175.279} C_VEL
LIN {X 0,Y 305.818,Z 1115.702,A -85,B 0,C 180,E1 15181.941,E2 15181.941} C_VEL
LIN {X 0,Y 299.102,Z 1131.901,A -85,B 0,C 180,E1 15189.244,E2 15189.244} C_VEL
LIN {X 0,Y 295.654,Z 1142.547,A -85,B 0,C 180,E1 15196.63,E2 15196.63} C_VEL
LIN {X 0,Y 294.205,Z 1148.364,A -85,B 0,C 180,E1 15204.091,E2 15204.091} C_VEL
LIN {X 0,Y 294.2,Z 1149.775,A -85,B 0,C 180,E1 15209.999,E2 15209.999} C_VEL
LIN {X 0,Y 294.207,Z 1148.31,A -85,B 0,C 180,E1 15215.907,E2 15215.907} C_VEL
LIN {X 0,Y 295.692,Z 1142.41,A -85,B 0,C 180,E1 15223.4,E2 15223.4} C_VEL
LIN {X 0,Y 299.64,Z 1130.394,A -85,B 0,C 180,E1 15231.49,E2 15231.49} C_VEL
LIN {X 0,Y 307.209,Z 1112.48,A -85,B 0,C 180,E1 15239.123,E2 15239.123} C_VEL
LIN {X 0,Y 317.067,Z 1091.031,A -85,B 0,C 180,E1 15245.408,E2 15245.408} C_VEL
LIN {X 0,Y 329.205,Z 1064.189,A -85,B 0,C 180,E1 15250.949,E2 15250.949} C_VEL
LIN {X 0,Y 341.618,Z 1033.872,A -85,B 0,C 180,E1 15255.39,E2 15255.39} C_VEL
LIN {X 0,Y 353.845,Z 998.993,A -85,B 0,C 180,E1 15258.953,E2 15258.953} C_VEL
LIN {X 0,Y 364.03,Z 962.114,A -85,B 0,C 180,E1 15261.519,E2 15261.519} C_VEL
LIN {X 0,Y 358.764,Z 944.716,A -85,B 0,C 180,E1 15264.483,E2 15264.483} C_VEL
LIN {X 0,Y 347.647,Z 920.348,A -85,B 0,C 180,E1 15269.736,E2 15269.736} C_VEL
LIN {X 0,Y 336.356,Z 900.348,A -85,B 0,C 180,E1 15275.381,E2 15275.381} C_VEL
LIN {X 0,Y 327.058,Z 886.817,A -85,B 0,C 180,E1 15280.927,E2 15280.927} C_VEL
LIN {X 0,Y 322.861,Z 880.679,A -85,B 0,C 180,E1 15284.185,E2 15284.185} C_VEL
LIN {X 0,Y 318.594,Z 874.153,A -85,B 0,C 180,E1 15288.697,E2 15288.697} C_VEL
LIN {X 0,Y 315.136,Z 869.79,A -85,B 0,C 180,E1 15297.248,E2 15297.248} C_VEL
LIN {X 0,Y 316.064,Z 871.729,A -85,B 0,C 180,E1 15302.747,E2 15302.747} C_VEL
LIN {X 0,Y 319.569,Z 875.487,A -85,B 0,C 180,E1 15308.086,E2 15308.086} C_VEL
LIN {X 0,Y 324.942,Z 883.691,A -85,B 0,C 180,E1 15313.13,E2 15313.13} C_VEL
LIN {X 0,Y 332.921,Z 895.279,A -85,B 0,C 180,E1 15318.391,E2 15318.391} C_VEL
LIN {X 0,Y 343.726,Z 913.936,A -85,B 0,C 180,E1 15324.217,E2 15324.217} C_VEL
LIN {X 0,Y 354.826,Z 937.321,A -85,B 0,C 180,E1 15329.621,E2 15329.621} C_VEL
LIN {X 0,Y 363.488,Z 963.196,A -85,B 0,C 180,E1 15334.306,E2 15334.306} C_VEL
LIN {X 0,Y 353.858,Z 1000.918,A -85,B 0,C 180,E1 15337.059,E2 15337.059} C_VEL
LIN {X 0,Y 342.158,Z 1036.297,A -85,B 0,C 180,E1 15340.593,E2 15340.593} C_VEL
LIN {X 0,Y 329.803,Z 1068.655,A -85,B 0,C 180,E1 15345.06,E2 15345.06} C_VEL
LIN {X 0,Y 317.941,Z 1097.648,A -85,B 0,C 180,E1 15350.57,E2 15350.57} C_VEL
LIN {X 0,Y 307.604,Z 1123.001,A -85,B 0,C 180,E1 15357.219,E2 15357.219} C_VEL
LIN {X 0,Y 300.334,Z 1142.712,A -85,B 0,C 180,E1 15364.406,E2 15364.406} C_VEL
LIN {X 0,Y 295.831,Z 1158.602,A -85,B 0,C 180,E1 15372.886,E2 15372.886} C_VEL
LIN {X 0,Y 294.395,Z 1166.473,A -85,B 0,C 180,E1 15379.631,E2 15379.631} C_VEL
LIN {X 0,Y 294.097,Z 1170.789,A -85,B 0,C 180,E1 15387.05,E2 15387.05} C_VEL
LIN {X 0,Y 294.033,Z 1170.787,A -85,B 0,C 180,E1 15392.953,E2 15392.953} C_VEL
LIN {X 0,Y 294.395,Z 1166.476,A -85,B 0,C 180,E1 15400.372,E2 15400.372} C_VEL
LIN {X 0,Y 296.066,Z 1157.418,A -85,B 0,C 180,E1 15407.871,E2 15407.871} C_VEL
LIN {X 0,Y 300.296,Z 1142.723,A -85,B 0,C 180,E1 15415.6,E2 15415.6} C_VEL
LIN {X 0,Y 308.488,Z 1120.805,A -85,B 0,C 180,E1 15423.455,E2 15423.455} C_VEL
LIN {X 0,Y 319.168,Z 1094.847,A -85,B 0,C 180,E1 15430.053,E2 15430.053} C_VEL
LIN {X 0,Y 331.581,Z 1064.449,A -85,B 0,C 180,E1 15435.621,E2 15435.621} C_VEL
LIN {X 0,Y 344.628,Z 1029.505,A -85,B 0,C 180,E1 15440.204,E2 15440.204} C_VEL
LIN {X 0,Y 344.947,Z 1028.598,A -85,B 0,C 180,E1 15440.297,E2 15440.297} C_VEL
LIN {X 0,Y 346.806,Z 1015.281,A -85,B 0,C 180,E1 15442.17,E2 15442.17} C_VEL
LIN {X 0,Y 348.146,Z 1003.431,A -85,B 0,C 180,E1 15443.759,E2 15443.759} C_VEL
LIN {X 0,Y 348.693,Z 1001.526,A -85,B 0,C 180,E1 15443.923,E2 15443.923} C_VEL
LIN {X 0,Y 358.137,Z 968.409,A -85,B 0,C 180,E1 15446.3,E2 15446.3} C_VEL
LIN {X 0,Y 357.458,Z 967.261,A -85,B 0,C 180,E1 15446.591,E2 15446.591} C_VEL
LIN {X 0,Y 337.982,Z 986.833,A -85,B 0,C 180,E1 15448.617,E2 15448.617} C_VEL
LIN {X 0,Y 317.607,Z 1002.601,A -85,B 0,C 180,E1 15451.53,E2 15451.53} C_VEL
LIN {X 0,Y 307.916,Z 1009.007,A -85,B 0,C 180,E1 15453.538,E2 15453.538} C_VEL
LIN {X 0,Y 302.784,Z 1030.247,A -85,B 0,C 180,E1 15457.595,E2 15457.595} C_VEL
LIN {X 0,Y 298.12,Z 1046.374,A -85,B 0,C 180,E1 15462.259,E2 15462.259} C_VEL
LIN {X 0,Y 294.305,Z 1057.381,A -85,B 0,C 180,E1 15467.37,E2 15467.37} C_VEL
LIN {X 0,Y 292.454,Z 1061.914,A -85,B 0,C 180,E1 15471.064,E2 15471.064} C_VEL
LIN {X 0,Y 290.551,Z 1064.231,A -85,B 0,C 180,E1 15477.012,E2 15477.012} C_VEL
LIN {X 0,Y 289.879,Z 1060.62,A -85,B 0,C 180,E1 15482.992,E2 15482.992} C_VEL
LIN {X 0,Y 290.336,Z 1050.944,A -85,B 0,C 180,E1 15488.999,E2 15488.999} C_VEL
LIN {X 0,Y 292.124,Z 1035.549,A -85,B 0,C 180,E1 15494.633,E2 15494.633} C_VEL
LIN {X 0,Y 294.788,Z 1015.609,A -85,B 0,C 180,E1 15499.499,E2 15499.499} C_VEL
LIN {X 0,Y 297.827,Z 995.079,A -85,B 0,C 180,E1 15503.199,E2 15503.199} C_VEL
LIN {X 0,Y 302.684,Z 992.089,A -85,B 0,C 180,E1 15504.669,E2 15504.669} C_VEL
LIN {X 0,Y 312.866,Z 983.588,A -85,B 0,C 180,E1 15506.977,E2 15506.977} C_VEL
LIN {X 0,Y 321.83,Z 975.767,A -85,B 0,C 180,E1 15508.757,E2 15508.757} C_VEL
LIN {X 0,Y 333.727,Z 963.295,A -85,B 0,C 180,E1 15510.686,E2 15510.686} C_VEL
LIN {X 0,Y 346.577,Z 946.853,A -85,B 0,C 180,E1 15512.425,E2 15512.425} C_VEL
LIN {X 0,Y 349.828,Z 941.461,A -85,B 0,C 180,E1 15512.748,E2 15512.748} C_VEL
LIN {X 0,Y 352.048,Z 944.408,A -85,B 0,C 180,E1 15513.66,E2 15513.66} C_VEL
LIN {X 0,Y 358.584,Z 963.546,A -85,B 0,C 180,E1 15517.315,E2 15517.315} C_VEL
LIN {X 0,Y 348.532,Z 1000.332,A -85,B 0,C 180,E1 15520.032,E2 15520.032} C_VEL
LIN {X 0,Y 335.966,Z 1034.899,A -85,B 0,C 180,E1 15523.62,E2 15523.62} C_VEL
LIN {X 0,Y 322.198,Z 1066.848,A -85,B 0,C 180,E1 15528.409,E2 15528.409} C_VEL
LIN {X 0,Y 309.071,Z 1094.469,A -85,B 0,C 180,E1 15534.424,E2 15534.424} C_VEL
LIN {X 0,Y 298.677,Z 1116.015,A -85,B 0,C 180,E1 15541.209,E2 15541.209} C_VEL
LIN {X 0,Y 291.586,Z 1132.201,A -85,B 0,C 180,E1 15548.684,E2 15548.684} C_VEL
LIN {X 0,Y 287.861,Z 1142.84,A -85,B 0,C 180,E1 15556.261,E2 15556.261} C_VEL
LIN {X 0,Y 286.317,Z 1148.653,A -85,B 0,C 180,E1 15563.927,E2 15563.927} C_VEL
LIN {X 0,Y 286.31,Z 1150.062,A -85,B 0,C 180,E1 15569.999,E2 15569.999} C_VEL
LIN {X 0,Y 286.319,Z 1148.599,A -85,B 0,C 180,E1 15576.07,E2 15576.07} C_VEL
LIN {X 0,Y 287.898,Z 1142.706,A -85,B 0,C 180,E1 15583.77,E2 15583.77} C_VEL
LIN {X 0,Y 292.127,Z 1130.703,A -85,B 0,C 180,E1 15592.071,E2 15592.071} C_VEL
LIN {X 0,Y 300.142,Z 1112.803,A -85,B 0,C 180,E1 15599.877,E2 15599.877} C_VEL
LIN {X 0,Y 310.794,Z 1090.836,A -85,B 0,C 180,E1 15606.399,E2 15606.399} C_VEL
LIN {X 0,Y 323.203,Z 1064.569,A -85,B 0,C 180,E1 15611.879,E2 15611.879} C_VEL
LIN {X 0,Y 336.558,Z 1033.077,A -85,B 0,C 180,E1 15616.504,E2 15616.504} C_VEL
LIN {X 0,Y 349.206,Z 997.876,A -85,B 0,C 180,E1 15620.075,E2 15620.075} C_VEL
LIN {X 0,Y 358.667,Z 963.725,A -85,B 0,C 180,E1 15622.529,E2 15622.529} C_VEL
LIN {X 0,Y 350.044,Z 939.497,A -85,B 0,C 180,E1 15627.275,E2 15627.275} C_VEL
LIN {X 0,Y 339.3,Z 917.182,A -85,B 0,C 180,E1 15632.796,E2 15632.796} C_VEL
LIN {X 0,Y 329.902,Z 901.141,A -85,B 0,C 180,E1 15638.193,E2 15638.193} C_VEL
LIN {X 0,Y 321.99,Z 888.756,A -85,B 0,C 180,E1 15644.002,E2 15644.002} C_VEL
LIN {X 0,Y 317.379,Z 881.87,A -85,B 0,C 180,E1 15649.002,E2 15649.002} C_VEL
LIN {X 0,Y 314.184,Z 877.726,A -85,B 0,C 180,E1 15658.621,E2 15658.621} C_VEL
LIN {X 0,Y 318.274,Z 883.188,A -85,B 0,C 180,E1 15667.775,E2 15667.775} C_VEL
LIN {X 0,Y 323.241,Z 891.191,A -85,B 0,C 180,E1 15672.77,E2 15672.77} C_VEL
LIN {X 0,Y 330.502,Z 902.292,A -85,B 0,C 180,E1 15677.926,E2 15677.926} C_VEL
LIN {X 0,Y 340.426,Z 920.358,A -85,B 0,C 180,E1 15683.682,E2 15683.682} C_VEL
LIN {X 0,Y 350.163,Z 941.938,A -85,B 0,C 180,E1 15688.853,E2 15688.853} C_VEL
LIN {X 0,Y 357.87,Z 965.902,A -85,B 0,C 180,E1 15693.365,E2 15693.365} C_VEL
LIN {X 0,Y 357.338,Z 970.886,A -85,B 0,C 180,E1 15693.849,E2 15693.849} C_VEL
LIN {X 0,Y 345.874,Z 1009.985,A -85,B 0,C 180,E1 15696.824,E2 15696.824} C_VEL
LIN {X 0,Y 332.904,Z 1046.253,A -85,B 0,C 180,E1 15700.82,E2 15700.82} C_VEL
LIN {X 0,Y 319.885,Z 1078.091,A -85,B 0,C 180,E1 15705.721,E2 15705.721} C_VEL
LIN {X 0,Y 307.424,Z 1106.744,A -85,B 0,C 180,E1 15711.862,E2 15711.862} C_VEL
LIN {X 0,Y 297.431,Z 1130.453,A -85,B 0,C 180,E1 15718.975,E2 15718.975} C_VEL
LIN {X 0,Y 290.56,Z 1149.217,A -85,B 0,C 180,E1 15726.995,E2 15726.995} C_VEL
LIN {X 0,Y 287.387,Z 1161.352,A -85,B 0,C 180,E1 15734.728,E2 15734.728} C_VEL
LIN {X 0,Y 286.362,Z 1167.46,A -85,B 0,C 180,E1 15740.874,E2 15740.874} C_VEL
LIN {X 0,Y 286.196,Z 1170.5,A -85,B 0,C 180,E1 15746.969,E2 15746.969} C_VEL
LIN {X 0,Y 286.142,Z 1170.5,A -85,B 0,C 180,E1 15753.035,E2 15753.035} C_VEL
LIN {X 0,Y 286.515,Z 1166.182,A -85,B 0,C 180,E1 15760.66,E2 15760.66} C_VEL
LIN {X 0,Y 288.345,Z 1157.113,A -85,B 0,C 180,E1 15768.366,E2 15768.366} C_VEL
LIN {X 0,Y 292.715,Z 1142.888,A -85,B 0,C 180,E1 15776.085,E2 15776.085} C_VEL
LIN {X 0,Y 301.158,Z 1121.617,A -85,B 0,C 180,E1 15783.979,E2 15783.979} C_VEL
LIN {X 0,Y 312.613,Z 1095.11,A -85,B 0,C 180,E1 15790.895,E2 15790.895} C_VEL
LIN {X 0,Y 325.92,Z 1063.953,A -85,B 0,C 180,E1 15796.666,E2 15796.666} C_VEL
LIN {X 0,Y 339.223,Z 1029.747,A -85,B 0,C 180,E1 15801.182,E2 15801.182} C_VEL
LIN {X 0,Y 348.693,Z 1001.526,A -85,B 0,C 180,E1 15803.923,E2 15803.923} C_VEL
LIN {X 0,Y 347.607,Z 997.299,A -85,B 0,C 180,E1 15804.791,E2 15804.791} C_VEL
LIN {X 0,Y 346.554,Z 993.035,A -85,B 0,C 180,E1 15805.657,E2 15805.657} C_VEL
LIN {X 0,Y 349.3,Z 983.863,A -85,B 0,C 180,E1 15806.322,E2 15806.322} C_VEL
LIN {X 0,Y 347.879,Z 983.87,A -85,B 0,C 180,E1 15806.646,E2 15806.646} C_VEL
LIN {X 0,Y 325.725,Z 1002.296,A -85,B 0,C 180,E1 15809.25,E2 15809.25} C_VEL
LIN {X 0,Y 305.64,Z 1014.986,A -85,B 0,C 180,E1 15812.61,E2 15812.61} C_VEL
LIN {X 0,Y 300.227,Z 1017.718,A -85,B 0,C 180,E1 15813.816,E2 15813.816} C_VEL
LIN {X 0,Y 294.895,Z 1036.863,A -85,B 0,C 180,E1 15818.013,E2 15818.013} C_VEL
LIN {X 0,Y 289.707,Z 1052.412,A -85,B 0,C 180,E1 15823.295,E2 15823.295} C_VEL
LIN {X 0,Y 286.347,Z 1060.549,A -85,B 0,C 180,E1 15827.789,E2 15827.789} C_VEL
LIN {X 0,Y 283.68,Z 1065.539,A -85,B 0,C 180,E1 15833.871,E2 15833.871} C_VEL
LIN {X 0,Y 282.315,Z 1064.543,A -85,B 0,C 180,E1 15839.999,E2 15839.999} C_VEL
LIN {X 0,Y 282.234,Z 1057.639,A -85,B 0,C 180,E1 15846.157,E2 15846.157} C_VEL
LIN {X 0,Y 283.234,Z 1045.304,A -85,B 0,C 180,E1 15851.953,E2 15851.953} C_VEL
LIN {X 0,Y 285.575,Z 1027.397,A -85,B 0,C 180,E1 15857.371,E2 15857.371} C_VEL
LIN {X 0,Y 288.681,Z 1006.075,A -85,B 0,C 180,E1 15861.918,E2 15861.918} C_VEL
LIN {X 0,Y 293.156,Z 1003.675,A -85,B 0,C 180,E1 15863.458,E2 15863.458} C_VEL
LIN {X 0,Y 310.232,Z 991.269,A -85,B 0,C 180,E1 15867.618,E2 15867.618} C_VEL
LIN {X 0,Y 322.7,Z 980.343,A -85,B 0,C 180,E1 15869.897,E2 15869.897} C_VEL
LIN {X 0,Y 334.32,Z 968.71,A -85,B 0,C 180,E1 15871.68,E2 15871.68} C_VEL
LIN {X 0,Y 347.622,Z 952.648,A -85,B 0,C 180,E1 15873.353,E2 15873.353} C_VEL
LIN {X 0,Y 349.147,Z 954.073,A -85,B 0,C 180,E1 15873.935,E2 15873.935} C_VEL
LIN {X 0,Y 353.121,Z 968.696,A -85,B 0,C 180,E1 15876.674,E2 15876.674} C_VEL
LIN {X 0,Y 341.884,Z 1005.504,A -85,B 0,C 180,E1 15879.44,E2 15879.44} C_VEL
LIN {X 0,Y 329.268,Z 1038.331,A -85,B 0,C 180,E1 15883.015,E2 15883.015} C_VEL
LIN {X 0,Y 315.4,Z 1068.913,A -85,B 0,C 180,E1 15887.769,E2 15887.769} C_VEL
LIN {X 0,Y 302.509,Z 1094.798,A -85,B 0,C 180,E1 15893.53,E2 15893.53} C_VEL
LIN {X 0,Y 291.595,Z 1116.326,A -85,B 0,C 180,E1 15900.441,E2 15900.441} C_VEL
LIN {X 0,Y 284.092,Z 1132.501,A -85,B 0,C 180,E1 15908.093,E2 15908.093} C_VEL
LIN {X 0,Y 280.075,Z 1143.218,A -85,B 0,C 180,E1 15915.964,E2 15915.964} C_VEL
LIN {X 0,Y 278.43,Z 1148.942,A -85,B 0,C 180,E1 15923.755,E2 15923.755} C_VEL
LIN {X 0,Y 278.412,Z 1150.349,A -85,B 0,C 180,E1 15929.999,E2 15929.999} C_VEL
LIN {X 0,Y 278.433,Z 1148.889,A -85,B 0,C 180,E1 15936.242,E2 15936.242} C_VEL
LIN {X 0,Y 280.145,Z 1142.964,A -85,B 0,C 180,E1 15944.195,E2 15944.195} C_VEL
LIN {X 0,Y 284.657,Z 1131.011,A -85,B 0,C 180,E1 15952.682,E2 15952.682} C_VEL
LIN {X 0,Y 293.154,Z 1113.125,A -85,B 0,C 180,E1 15960.665,E2 15960.665} C_VEL
LIN {X 0,Y 304.156,Z 1091.534,A -85,B 0,C 180,E1 15967.214,E2 15967.214} C_VEL
LIN {X 0,Y 317.275,Z 1064.95,A -85,B 0,C 180,E1 15972.846,E2 15972.846} C_VEL
LIN {X 0,Y 331.1,Z 1033.594,A -85,B 0,C 180,E1 15977.494,E2 15977.494} C_VEL
LIN {X 0,Y 344.185,Z 998.421,A -85,B 0,C 180,E1 15981.086,E2 15981.086} C_VEL
LIN {X 0,Y 353.19,Z 967.031,A -85,B 0,C 180,E1 15983.399,E2 15983.399} C_VEL
LIN {X 0,Y 345.133,Z 943.414,A -85,B 0,C 180,E1 15988.24,E2 15988.24} C_VEL
LIN {X 0,Y 335.17,Z 921.912,A -85,B 0,C 180,E1 15993.875,E2 15993.875} C_VEL
LIN {X 0,Y 326.972,Z 907.499,A -85,B 0,C 180,E1 15999.019,E2 15999.019} C_VEL
LIN {X 0,Y 320.298,Z 896.201,A -85,B 0,C 180,E1 16004.437,E2 16004.437} C_VEL
LIN {X 0,Y 316.036,Z 889.586,A -85,B 0,C 180,E1 16009.304,E2 16009.304} C_VEL
LIN {X 0,Y 313.163,Z 885.56,A -85,B 0,C 180,E1 16018.616,E2 16018.616} C_VEL
LIN {X 0,Y 316.899,Z 890.929,A -85,B 0,C 180,E1 16027.551,E2 16027.551} C_VEL
LIN {X 0,Y 321.535,Z 898.831,A -85,B 0,C 180,E1 16032.493,E2 16032.493} C_VEL
LIN {X 0,Y 328.514,Z 910.325,A -85,B 0,C 180,E1 16037.778,E2 16037.778} C_VEL
LIN {X 0,Y 337.439,Z 927.6,A -85,B 0,C 180,E1 16043.378,E2 16043.378} C_VEL
LIN {X 0,Y 346.598,Z 949.683,A -85,B 0,C 180,E1 16048.718,E2 16048.718} C_VEL
LIN {X 0,Y 352.604,Z 971.272,A -85,B 0,C 180,E1 16052.826,E2 16052.826} C_VEL
LIN {X 0,Y 340.808,Z 1010.216,A -85,B 0,C 180,E1 16055.803,E2 16055.803} C_VEL
LIN {X 0,Y 327.845,Z 1045.265,A -85,B 0,C 180,E1 16059.663,E2 16059.663} C_VEL
LIN {X 0,Y 313.98,Z 1077.867,A -85,B 0,C 180,E1 16064.703,E2 16064.703} C_VEL
LIN {X 0,Y 301.264,Z 1105.795,A -85,B 0,C 180,E1 16070.733,E2 16070.733} C_VEL
LIN {X 0,Y 290.797,Z 1129.144,A -85,B 0,C 180,E1 16077.766,E2 16077.766} C_VEL
LIN {X 0,Y 283.45,Z 1147.739,A -85,B 0,C 180,E1 16085.732,E2 16085.732} C_VEL
LIN {X 0,Y 279.61,Z 1161.05,A -85,B 0,C 180,E1 16094.292,E2 16094.292} C_VEL
LIN {X 0,Y 278.475,Z 1167.166,A -85,B 0,C 180,E1 16100.614,E2 16100.614} C_VEL
LIN {X 0,Y 278.285,Z 1170.212,A -85,B 0,C 180,E1 16106.882,E2 16106.882} C_VEL
LIN {X 0,Y 278.233,Z 1170.212,A -85,B 0,C 180,E1 16113.121,E2 16113.121} C_VEL
LIN {X 0,Y 278.636,Z 1166.019,A -85,B 0,C 180,E1 16120.804,E2 16120.804} C_VEL
LIN {X 0,Y 280.658,Z 1156.808,A -85,B 0,C 180,E1 16128.888,E2 16128.888} C_VEL
LIN {X 0,Y 285.353,Z 1142.572,A -85,B 0,C 180,E1 16136.811,E2 16136.811} C_VEL
LIN {X 0,Y 294.339,Z 1121.184,A -85,B 0,C 180,E1 16144.912,E2 16144.912} C_VEL
LIN {X 0,Y 306.754,Z 1093.811,A -85,B 0,C 180,E1 16152.118,E2 16152.118} C_VEL
LIN {X 0,Y 320.539,Z 1063.006,A -85,B 0,C 180,E1 16157.821,E2 16157.821} C_VEL
LIN {X 0,Y 334.546,Z 1028.085,A -85,B 0,C 180,E1 16162.408,E2 16162.408} C_VEL
LIN {X 0,Y 346.554,Z 993.035,A -85,B 0,C 180,E1 16165.657,E2 16165.657} C_VEL
LIN {X 0,Y 344.406,Z 992.499,A -85,B 0,C 180,E1 16166.227,E2 16166.227} C_VEL
LIN {X 0,Y 335.54,Z 999.688,A -85,B 0,C 180,E1 16167.175,E2 16167.175} C_VEL
LIN {X 0,Y 329.929,Z 1004.654,A -85,B 0,C 180,E1 16167.734,E2 16167.734} C_VEL
LIN {X 0,Y 309.339,Z 1018.171,A -85,B 0,C 180,E1 16170.697,E2 16170.697} C_VEL
LIN {X 0,Y 292.212,Z 1026.685,A -85,B 0,C 180,E1 16174.283,E2 16174.283} C_VEL
LIN {X 0,Y 286.254,Z 1045.004,A -85,B 0,C 180,E1 16179.083,E2 16179.083} C_VEL
LIN {X 0,Y 281.201,Z 1057.845,A -85,B 0,C 180,E1 16184.382,E2 16184.382} C_VEL
LIN {X 0,Y 277.814,Z 1064.728,A -85,B 0,C 180,E1 16189.419,E2 16189.419} C_VEL
LIN {X 0,Y 276.009,Z 1067.237,A -85,B 0,C 180,E1 16193.7,E2 16193.7} C_VEL
LIN {X 0,Y 274.553,Z 1065.911,A -85,B 0,C 180,E1 16199.999,E2 16199.999} C_VEL
LIN {X 0,Y 274.451,Z 1058.659,A -85,B 0,C 180,E1 16206.333,E2 16206.333} C_VEL
LIN {X 0,Y 275.521,Z 1045.988,A -85,B 0,C 180,E1 16212.292,E2 16212.292} C_VEL
LIN {X 0,Y 277.979,Z 1027.582,A -85,B 0,C 180,E1 16217.861,E2 16217.861} C_VEL
LIN {X 0,Y 279.824,Z 1015.959,A -85,B 0,C 180,E1 16220.588,E2 16220.588} C_VEL
LIN {X 0,Y 283.154,Z 1014.595,A -85,B 0,C 180,E1 16221.978,E2 16221.978} C_VEL
LIN {X 0,Y 299.367,Z 1004.268,A -85,B 0,C 180,E1 16226.49,E2 16226.49} C_VEL
LIN {X 0,Y 319.866,Z 988.574,A -85,B 0,C 180,E1 16230.499,E2 16230.499} C_VEL
LIN {X 0,Y 335.693,Z 973.231,A -85,B 0,C 180,E1 16232.763,E2 16232.763} C_VEL
LIN {X 0,Y 344.467,Z 963.505,A -85,B 0,C 180,E1 16233.832,E2 16233.832} C_VEL
LIN {X 0,Y 346.119,Z 964.579,A -85,B 0,C 180,E1 16234.401,E2 16234.401} C_VEL
LIN {X 0,Y 347.744,Z 972.013,A -85,B 0,C 180,E1 16235.803,E2 16235.803} C_VEL
LIN {X 0,Y 336.338,Z 1007.512,A -85,B 0,C 180,E1 16238.536,E2 16238.536} C_VEL
LIN {X 0,Y 323.445,Z 1039.684,A -85,B 0,C 180,E1 16242.108,E2 16242.108} C_VEL
LIN {X 0,Y 309.487,Z 1069.269,A -85,B 0,C 180,E1 16246.768,E2 16246.768} C_VEL
LIN {X 0,Y 296.065,Z 1095.123,A -85,B 0,C 180,E1 16252.603,E2 16252.603} C_VEL
LIN {X 0,Y 284.571,Z 1116.637,A -85,B 0,C 180,E1 16259.636,E2 16259.636} C_VEL
LIN {X 0,Y 276.617,Z 1132.8,A -85,B 0,C 180,E1 16267.469,E2 16267.469} C_VEL
LIN {X 0,Y 272.31,Z 1143.468,A -85,B 0,C 180,E1 16275.508,E2 16275.508} C_VEL
LIN {X 0,Y 270.545,Z 1149.231,A -85,B 0,C 180,E1 16283.572,E2 16283.572} C_VEL
LIN {X 0,Y 270.537,Z 1150.636,A -85,B 0,C 180,E1 16289.999,E2 16289.999} C_VEL
LIN {X 0,Y 270.547,Z 1149.179,A -85,B 0,C 180,E1 16296.425,E2 16296.425} C_VEL
LIN {X 0,Y 272.337,Z 1143.376,A -85,B 0,C 180,E1 16304.487,E2 16304.487} C_VEL
LIN {X 0,Y 277.239,Z 1131.317,A -85,B 0,C 180,E1 16313.324,E2 16313.324} C_VEL
LIN {X 0,Y 286.211,Z 1113.445,A -85,B 0,C 180,E1 16321.493,E2 16321.493} C_VEL
LIN {X 0,Y 297.783,Z 1091.876,A -85,B 0,C 180,E1 16328.151,E2 16328.151} C_VEL
LIN {X 0,Y 311.447,Z 1065.326,A -85,B 0,C 180,E1 16333.849,E2 16333.849} C_VEL
LIN {X 0,Y 325.781,Z 1034.064,A -85,B 0,C 180,E1 16338.518,E2 16338.518} C_VEL
LIN {X 0,Y 339.271,Z 998.969,A -85,B 0,C 180,E1 16342.125,E2 16342.125} C_VEL
LIN {X 0,Y 347.739,Z 970.393,A -85,B 0,C 180,E1 16344.288,E2 16344.288} C_VEL
LIN {X 0,Y 340.276,Z 947.542,A -85,B 0,C 180,E1 16349.221,E2 16349.221} C_VEL
LIN {X 0,Y 331.123,Z 926.508,A -85,B 0,C 180,E1 16354.982,E2 16354.982} C_VEL
LIN {X 0,Y 322.14,Z 909.879,A -85,B 0,C 180,E1 16361.44,E2 16361.44} C_VEL
LIN {X 0,Y 317.35,Z 902.45,A -85,B 0,C 180,E1 16365.862,E2 16365.862} C_VEL
LIN {X 0,Y 314.466,Z 897.129,A -85,B 0,C 180,E1 16369.883,E2 16369.883} C_VEL
LIN {X 0,Y 312.024,Z 893.377,A -85,B 0,C 180,E1 16378.611,E2 16378.611} C_VEL
LIN {X 0,Y 315.376,Z 898.548,A -85,B 0,C 180,E1 16387.24,E2 16387.24} C_VEL
LIN {X 0,Y 319.797,Z 906.726,A -85,B 0,C 180,E1 16392.388,E2 16392.388} C_VEL
LIN {X 0,Y 325.906,Z 917.509,A -85,B 0,C 180,E1 16397.401,E2 16397.401} C_VEL
LIN {X 0,Y 334.005,Z 934.102,A -85,B 0,C 180,E1 16402.892,E2 16402.892} C_VEL
LIN {X 0,Y 342.287,Z 955.533,A -85,B 0,C 180,E1 16408.209,E2 16408.209} C_VEL
LIN {X 0,Y 347.098,Z 974.929,A -85,B 0,C 180,E1 16411.985,E2 16411.985} C_VEL
LIN {X 0,Y 335.087,Z 1012.484,A -85,B 0,C 180,E1 16414.931,E2 16414.931} C_VEL
LIN {X 0,Y 321.297,Z 1048.01,A -85,B 0,C 180,E1 16418.963,E2 16418.963} C_VEL
LIN {X 0,Y 307.501,Z 1078.987,A -85,B 0,C 180,E1 16423.894,E2 16423.894} C_VEL
LIN {X 0,Y 294.127,Z 1106.967,A -85,B 0,C 180,E1 16430.121,E2 16430.121} C_VEL
LIN {X 0,Y 282.904,Z 1130.815,A -85,B 0,C 180,E1 16437.643,E2 16437.643} C_VEL
LIN {X 0,Y 275.4,Z 1148.987,A -85,B 0,C 180,E1 16445.89,E2 16445.89} C_VEL
LIN {X 0,Y 271.825,Z 1160.748,A -85,B 0,C 180,E1 16453.83,E2 16453.83} C_VEL
LIN {X 0,Y 270.593,Z 1166.872,A -85,B 0,C 180,E1 16460.338,E2 16460.338} C_VEL
LIN {X 0,Y 270.39,Z 1169.924,A -85,B 0,C 180,E1 16466.791,E2 16466.791} C_VEL
LIN {X 0,Y 270.345,Z 1169.924,A -85,B 0,C 180,E1 16473.212,E2 16473.212} C_VEL
LIN {X 0,Y 270.775,Z 1165.857,A -85,B 0,C 180,E1 16480.956,E2 16480.956} C_VEL
LIN {X 0,Y 272.968,Z 1156.479,A -85,B 0,C 180,E1 16489.459,E2 16489.459} C_VEL
LIN {X 0,Y 278.038,Z 1142.256,A -85,B 0,C 180,E1 16497.575,E2 16497.575} C_VEL
LIN {X 0,Y 287.646,Z 1120.85,A -85,B 0,C 180,E1 16505.848,E2 16505.848} C_VEL
LIN {X 0,Y 299.794,Z 1095.375,A -85,B 0,C 180,E1 16512.751,E2 16512.751} C_VEL
LIN {X 0,Y 314.583,Z 1063.674,A -85,B 0,C 180,E1 16518.77,E2 16518.77} C_VEL
LIN {X 0,Y 329.092,Z 1029.001,A -85,B 0,C 180,E1 16523.387,E2 16523.387} C_VEL
LIN {X 0,Y 340.551,Z 996.29,A -85,B 0,C 180,E1 16526.525,E2 16526.525} C_VEL
LIN {X 0,Y 329.929,Z 1004.654,A -85,B 0,C 180,E1 16527.734,E2 16527.734} C_VEL
LIN {X 0,Y 314.685,Z 1020.001,A -85,B 0,C 180,E1 16528.732,E2 16528.732} C_VEL
LIN {X 0,Y 313.649,Z 1020.609,A -85,B 0,C 180,E1 16528.881,E2 16528.881} C_VEL
LIN {X 0,Y 293.9,Z 1030.972,A -85,B 0,C 180,E1 16532.378,E2 16532.378} C_VEL
LIN {X 0,Y 284.077,Z 1034.968,A -85,B 0,C 180,E1 16534.762,E2 16534.762} C_VEL
LIN {X 0,Y 277.655,Z 1052.003,A -85,B 0,C 180,E1 16540.074,E2 16540.074} C_VEL
LIN {X 0,Y 272.686,Z 1062.653,A -85,B 0,C 180,E1 16545.531,E2 16545.531} C_VEL
LIN {X 0,Y 269.752,Z 1067.57,A -85,B 0,C 180,E1 16550.305,E2 16550.305} C_VEL
LIN {X 0,Y 267.375,Z 1068.847,A -85,B 0,C 180,E1 16556.753,E2 16556.753} C_VEL
LIN {X 0,Y 266.526,Z 1064.236,A -85,B 0,C 180,E1 16563.255,E2 16563.255} C_VEL
LIN {X 0,Y 266.894,Z 1055.181,A -85,B 0,C 180,E1 16568.973,E2 16568.973} C_VEL
LIN {X 0,Y 268.795,Z 1039.381,A -85,B 0,C 180,E1 16575.098,E2 16575.098} C_VEL
LIN {X 0,Y 270.744,Z 1025.24,A -85,B 0,C 180,E1 16578.972,E2 16578.972} C_VEL
LIN {X 0,Y 273.562,Z 1024.286,A -85,B 0,C 180,E1 16580.396,E2 16580.396} C_VEL
LIN {X 0,Y 294.511,Z 1012.269,A -85,B 0,C 180,E1 16586.729,E2 16586.729} C_VEL
LIN {X 0,Y 315.843,Z 997.167,A -85,B 0,C 180,E1 16590.93,E2 16590.93} C_VEL
LIN {X 0,Y 335.028,Z 980.019,A -85,B 0,C 180,E1 16593.61,E2 16593.61} C_VEL
LIN {X 0,Y 341.897,Z 972.496,A -85,B 0,C 180,E1 16594.371,E2 16594.371} C_VEL
LIN {X 0,Y 341.937,Z 977.266,A -85,B 0,C 180,E1 16595.037,E2 16595.037} C_VEL
LIN {X 0,Y 328.587,Z 1015.409,A -85,B 0,C 180,E1 16598.162,E2 16598.162} C_VEL
LIN {X 0,Y 314.71,Z 1047.661,A -85,B 0,C 180,E1 16602.089,E2 16602.089} C_VEL
LIN {X 0,Y 299.566,Z 1077.499,A -85,B 0,C 180,E1 16607.306,E2 16607.306} C_VEL
LIN {X 0,Y 285.445,Z 1103.096,A -85,B 0,C 180,E1 16613.881,E2 16613.881} C_VEL
LIN {X 0,Y 274.892,Z 1122.029,A -85,B 0,C 180,E1 16620.963,E2 16620.963} C_VEL
LIN {X 0,Y 267.352,Z 1136.917,A -85,B 0,C 180,E1 16629.315,E2 16629.315} C_VEL
LIN {X 0,Y 263.876,Z 1145.692,A -85,B 0,C 180,E1 16637.243,E2 16637.243} C_VEL
LIN {X 0,Y 262.662,Z 1149.52,A -85,B 0,C 180,E1 16643.378,E2 16643.378} C_VEL
LIN {X 0,Y 262.638,Z 1150.923,A -85,B 0,C 180,E1 16649.998,E2 16649.998} C_VEL
LIN {X 0,Y 262.664,Z 1149.469,A -85,B 0,C 180,E1 16656.619,E2 16656.619} C_VEL
LIN {X 0,Y 264.597,Z 1143.669,A -85,B 0,C 180,E1 16664.921,E2 16664.921} C_VEL
LIN {X 0,Y 269.835,Z 1131.623,A -85,B 0,C 180,E1 16674.004,E2 16674.004} C_VEL
LIN {X 0,Y 279.359,Z 1113.763,A -85,B 0,C 180,E1 16682.358,E2 16682.358} C_VEL
LIN {X 0,Y 292.118,Z 1091.073,A -85,B 0,C 180,E1 16689.415,E2 16689.415} C_VEL
LIN {X 0,Y 306.654,Z 1063.825,A -85,B 0,C 180,E1 16695.215,E2 16695.215} C_VEL
LIN {X 0,Y 321.309,Z 1032.776,A -85,B 0,C 180,E1 16699.789,E2 16699.789} C_VEL
LIN {X 0,Y 335.04,Z 997.834,A -85,B 0,C 180,E1 16703.336,E2 16703.336} C_VEL
LIN {X 0,Y 342.489,Z 974.151,A -85,B 0,C 180,E1 16705.12,E2 16705.12} C_VEL
LIN {X 0,Y 335.535,Z 951.508,A -85,B 0,C 180,E1 16710.244,E2 16710.244} C_VEL
LIN {X 0,Y 326.981,Z 931.36,A -85,B 0,C 180,E1 16716.102,E2 16716.102} C_VEL
LIN {X 0,Y 319.443,Z 916.694,A -85,B 0,C 180,E1 16722.111,E2 16722.111} C_VEL
LIN {X 0,Y 315.391,Z 909.794,A -85,B 0,C 180,E1 16726.318,E2 16726.318} C_VEL
LIN {X 0,Y 312.8,Z 904.808,A -85,B 0,C 180,E1 16730.138,E2 16730.138} C_VEL
LIN {X 0,Y 310.685,Z 901.154,A -85,B 0,C 180,E1 16738.605,E2 16738.605} C_VEL
LIN {X 0,Y 313.625,Z 906.074,A -85,B 0,C 180,E1 16746.933,E2 16746.933} C_VEL
LIN {X 0,Y 317.798,Z 914.432,A -85,B 0,C 180,E1 16752.205,E2 16752.205} C_VEL
LIN {X 0,Y 323.714,Z 925.601,A -85,B 0,C 180,E1 16757.374,E2 16757.374} C_VEL
LIN {X 0,Y 331.156,Z 942.132,A -85,B 0,C 180,E1 16762.865,E2 16762.865} C_VEL
LIN {X 0,Y 338.997,Z 965.089,A -85,B 0,C 180,E1 16768.508,E2 16768.508} C_VEL
LIN {X 0,Y 341.79,Z 978.173,A -85,B 0,C 180,E1 16771.092,E2 16771.092} C_VEL
LIN {X 0,Y 328.461,Z 1017.588,A -85,B 0,C 180,E1 16774.309,E2 16774.309} C_VEL
LIN {X 0,Y 313.139,Z 1054.57,A -85,B 0,C 180,E1 16778.769,E2 16778.769} C_VEL
LIN {X 0,Y 298.054,Z 1086.325,A -85,B 0,C 180,E1 16784.274,E2 16784.274} C_VEL
LIN {X 0,Y 283.929,Z 1114.242,A -85,B 0,C 180,E1 16791.202,E2 16791.202} C_VEL
LIN {X 0,Y 272.995,Z 1136.942,A -85,B 0,C 180,E1 16799.368,E2 16799.368} C_VEL
LIN {X 0,Y 266.11,Z 1153.768,A -85,B 0,C 180,E1 16808.296,E2 16808.296} C_VEL
LIN {X 0,Y 263.22,Z 1163.904,A -85,B 0,C 180,E1 16816.699,E2 16816.699} C_VEL
LIN {X 0,Y 262.426,Z 1168.483,A -85,B 0,C 180,E1 16823.375,E2 16823.375} C_VEL
LIN {X 0,Y 262.63,Z 1170.025,A -85,B 0,C 180,E1 16830.002,E2 16830.002} C_VEL
LIN {X 0,Y 262.423,Z 1168.488,A -85,B 0,C 180,E1 16836.628,E2 16836.628} C_VEL
LIN {X 0,Y 263.604,Z 1162.257,A -85,B 0,C 180,E1 16844.981,E2 16844.981} C_VEL
LIN {X 0,Y 266.998,Z 1151.113,A -85,B 0,C 180,E1 16853.39,E2 16853.39} C_VEL
LIN {X 0,Y 274.217,Z 1134.332,A -85,B 0,C 180,E1 16861.753,E2 16861.753} C_VEL
LIN {X 0,Y 285.345,Z 1111.667,A -85,B 0,C 180,E1 16869.552,E2 16869.552} C_VEL
LIN {X 0,Y 299.342,Z 1083.711,A -85,B 0,C 180,E1 16876.273,E2 16876.273} C_VEL
LIN {X 0,Y 314.608,Z 1051.215,A -85,B 0,C 180,E1 16881.73,E2 16881.73} C_VEL
LIN {X 0,Y 329.246,Z 1015.726,A -85,B 0,C 180,E1 16885.874,E2 16885.874} C_VEL
LIN {X 0,Y 331.604,Z 1008.82,A -85,B 0,C 180,E1 16886.563,E2 16886.563} C_VEL
LIN {X 0,Y 313.649,Z 1020.609,A -85,B 0,C 180,E1 16888.881,E2 16888.881} C_VEL
LIN {X 0,Y 305.091,Z 1027.875,A -85,B 0,C 180,E1 16889.649,E2 16889.649} C_VEL
LIN {X 0,Y 297.059,Z 1034.39,A -85,B 0,C 180,E1 16890.39,E2 16890.39} C_VEL
LIN {X 0,Y 296.56,Z 1034.613,A -85,B 0,C 180,E1 16890.484,E2 16890.484} C_VEL
LIN {X 0,Y 276.241,Z 1042.661,A -85,B 0,C 180,E1 16895.209,E2 16895.209} C_VEL
LIN {X 0,Y 269,Z 1058.168,A -85,B 0,C 180,E1 16901.117,E2 16901.117} C_VEL
LIN {X 0,Y 264.097,Z 1066.832,A -85,B 0,C 180,E1 16906.743,E2 16906.743} C_VEL
LIN {X 0,Y 260.71,Z 1070.662,A -85,B 0,C 180,E1 16913.329,E2 16913.329} C_VEL
LIN {X 0,Y 259.009,Z 1068.628,A -85,B 0,C 180,E1 16919.998,E2 16919.998} C_VEL
LIN {X 0,Y 258.899,Z 1060.651,A -85,B 0,C 180,E1 16926.715,E2 16926.715} C_VEL
LIN {X 0,Y 260.086,Z 1047.101,A -85,B 0,C 180,E1 16933.034,E2 16933.034} C_VEL
LIN {X 0,Y 262.124,Z 1033.847,A -85,B 0,C 180,E1 16937.424,E2 16937.424} C_VEL
LIN {X 0,Y 271.454,Z 1029.561,A -85,B 0,C 180,E1 16941.581,E2 16941.581} C_VEL
LIN {X 0,Y 290.117,Z 1019.421,A -85,B 0,C 180,E1 16947.071,E2 16947.071} C_VEL
LIN {X 0,Y 307.818,Z 1008.053,A -85,B 0,C 180,E1 16950.681,E2 16950.681} C_VEL
LIN {X 0,Y 329.643,Z 991.03,A -85,B 0,C 180,E1 16953.92,E2 16953.92} C_VEL
LIN {X 0,Y 334.324,Z 986.606,A -85,B 0,C 180,E1 16954.475,E2 16954.475} C_VEL
LIN {X 0,Y 321.218,Z 1021.899,A -85,B 0,C 180,E1 16957.692,E2 16957.692} C_VEL
LIN {X 0,Y 305.838,Z 1055.032,A -85,B 0,C 180,E1 16962.043,E2 16962.043} C_VEL
LIN {X 0,Y 290.813,Z 1083.02,A -85,B 0,C 180,E1 16967.4,E2 16967.4} C_VEL
LIN {X 0,Y 276.831,Z 1107.02,A -85,B 0,C 180,E1 16974.082,E2 16974.082} C_VEL
LIN {X 0,Y 265.412,Z 1126.621,A -85,B 0,C 180,E1 16982.217,E2 16982.217} C_VEL
LIN {X 0,Y 258.405,Z 1140.431,A -85,B 0,C 180,E1 16991.198,E2 16991.198} C_VEL
LIN {X 0,Y 255.374,Z 1148.034,A -85,B 0,C 180,E1 16999.753,E2 16999.753} C_VEL
LIN {X 0,Y 254.636,Z 1150.866,A -85,B 0,C 180,E1 17006.589,E2 17006.589} C_VEL
LIN {X 0,Y 254.653,Z 1150.836,A -85,B 0,C 180,E1 17013.407,E2 17013.407} C_VEL
LIN {X 0,Y 255.709,Z 1147.117,A -85,B 0,C 180,E1 17021.508,E2 17021.508} C_VEL
LIN {X 0,Y 259.366,Z 1138.114,A -85,B 0,C 180,E1 17030.502,E2 17030.502} C_VEL
LIN {X 0,Y 266.815,Z 1124.082,A -85,B 0,C 180,E1 17038.915,E2 17038.915} C_VEL
LIN {X 0,Y 277.829,Z 1105.352,A -85,B 0,C 180,E1 17046.345,E2 17046.345} C_VEL
LIN {X 0,Y 291.832,Z 1081.072,A -85,B 0,C 180,E1 17052.929,E2 17052.929} C_VEL
LIN {X 0,Y 306.917,Z 1052.657,A -85,B 0,C 180,E1 17058.222,E2 17058.222} C_VEL
LIN {X 0,Y 321.528,Z 1021.157,A -85,B 0,C 180,E1 17062.259,E2 17062.259} C_VEL
LIN {X 0,Y 334.502,Z 986.46,A -85,B 0,C 180,E1 17065.372,E2 17065.372} C_VEL
LIN {X 0,Y 337.089,Z 978.784,A -85,B 0,C 180,E1 17065.891,E2 17065.891} C_VEL
LIN {X 0,Y 332.047,Z 959.607,A -85,B 0,C 180,E1 17070.235,E2 17070.235} C_VEL
LIN {X 0,Y 324.701,Z 939.872,A -85,B 0,C 180,E1 17075.924,E2 17075.924} C_VEL
LIN {X 0,Y 317.196,Z 924.095,A -85,B 0,C 180,E1 17082.381,E2 17082.381} C_VEL
LIN {X 0,Y 313.162,Z 916.929,A -85,B 0,C 180,E1 17086.835,E2 17086.835} C_VEL
LIN {X 0,Y 311.008,Z 912.367,A -85,B 0,C 180,E1 17090.515,E2 17090.515} C_VEL
LIN {X 0,Y 309.193,Z 908.911,A -85,B 0,C 180,E1 17098.598,E2 17098.598} C_VEL
LIN {X 0,Y 311.781,Z 913.753,A -85,B 0,C 180,E1 17106.711,E2 17106.711} C_VEL
LIN {X 0,Y 315.65,Z 922.047,A -85,B 0,C 180,E1 17112.026,E2 17112.026} C_VEL
LIN {X 0,Y 322.136,Z 935.104,A -85,B 0,C 180,E1 17118.039,E2 17118.039} C_VEL
LIN {X 0,Y 330.021,Z 955.82,A -85,B 0,C 180,E1 17124.386,E2 17124.386} C_VEL
LIN {X 0,Y 335.866,Z 977.055,A -85,B 0,C 180,E1 17129.355,E2 17129.355} C_VEL
LIN {X 0,Y 336.35,Z 981.834,A -85,B 0,C 180,E1 17130.213,E2 17130.213} C_VEL
LIN {X 0,Y 322.465,Z 1020.703,A -85,B 0,C 180,E1 17133.484,E2 17133.484} C_VEL
LIN {X 0,Y 307.015,Z 1056.317,A -85,B 0,C 180,E1 17137.902,E2 17137.902} C_VEL
LIN {X 0,Y 291.677,Z 1087.217,A -85,B 0,C 180,E1 17143.387,E2 17143.387} C_VEL
LIN {X 0,Y 277.329,Z 1114.329,A -85,B 0,C 180,E1 17150.269,E2 17150.269} C_VEL
LIN {X 0,Y 266.228,Z 1136.003,A -85,B 0,C 180,E1 17158.173,E2 17158.173} C_VEL
LIN {X 0,Y 258.97,Z 1152.188,A -85,B 0,C 180,E1 17166.757,E2 17166.757} C_VEL
LIN {X 0,Y 255.815,Z 1161.952,A -85,B 0,C 180,E1 17174.555,E2 17174.555} C_VEL
LIN {X 0,Y 254.542,Z 1168.193,A -85,B 0,C 180,E1 17183.169,E2 17183.169} C_VEL
LIN {X 0,Y 254.754,Z 1169.738,A -85,B 0,C 180,E1 17190.002,E2 17190.002} C_VEL
LIN {X 0,Y 254.54,Z 1168.198,A -85,B 0,C 180,E1 17196.834,E2 17196.834} C_VEL
LIN {X 0,Y 255.813,Z 1161.961,A -85,B 0,C 180,E1 17205.449,E2 17205.449} C_VEL
LIN {X 0,Y 259.494,Z 1150.806,A -85,B 0,C 180,E1 17214.109,E2 17214.109} C_VEL
LIN {X 0,Y 267.097,Z 1134.136,A -85,B 0,C 180,E1 17222.642,E2 17222.642} C_VEL
LIN {X 0,Y 278.998,Z 1111.326,A -85,B 0,C 180,E1 17230.637,E2 17230.637} C_VEL
LIN {X 0,Y 293.846,Z 1083.074,A -85,B 0,C 180,E1 17237.486,E2 17237.486} C_VEL
LIN {X 0,Y 309.603,Z 1050.795,A -85,B 0,C 180,E1 17242.92,E2 17242.92} C_VEL
LIN {X 0,Y 322.275,Z 1020.544,A -85,B 0,C 180,E1 17246.631,E2 17246.631} C_VEL
LIN {X 0,Y 297.536,Z 1034.216,A -85,B 0,C 180,E1 17250.289,E2 17250.289} C_VEL
LIN {X 0,Y 296.56,Z 1034.613,A -85,B 0,C 180,E1 17250.484,E2 17250.484} C_VEL
LIN {X 0,Y 287.918,Z 1040.711,A -85,B 0,C 180,E1 17251.559,E2 17251.559} C_VEL
LIN {X 0,Y 280.251,Z 1046.084,A -85,B 0,C 180,E1 17252.47,E2 17252.47} C_VEL
LIN {X 0,Y 279.285,Z 1046.487,A -85,B 0,C 180,E1 17252.681,E2 17252.681} C_VEL
LIN {X 0,Y 267.29,Z 1050.508,A -85,B 0,C 180,E1 17256.197,E2 17256.197} C_VEL
LIN {X 0,Y 260.301,Z 1063.665,A -85,B 0,C 180,E1 17262.219,E2 17262.219} C_VEL
LIN {X 0,Y 255.935,Z 1069.996,A -85,B 0,C 180,E1 17267.487,E2 17267.487} C_VEL
LIN {X 0,Y 253.054,Z 1072.395,A -85,B 0,C 180,E1 17273.126,E2 17273.126} C_VEL
LIN {X 0,Y 251.225,Z 1069.971,A -85,B 0,C 180,E1 17279.998,E2 17279.998} C_VEL
LIN {X 0,Y 251.092,Z 1061.553,A -85,B 0,C 180,E1 17286.924,E2 17286.924} C_VEL
LIN {X 0,Y 252.403,Z 1047.53,A -85,B 0,C 180,E1 17293.438,E2 17293.438} C_VEL
LIN {X 0,Y 253.394,Z 1042.036,A -85,B 0,C 180,E1 17295.595,E2 17295.595} C_VEL
LIN {X 0,Y 268.085,Z 1035.542,A -85,B 0,C 180,E1 17302.406,E2 17302.406} C_VEL
LIN {X 0,Y 288.575,Z 1024.975,A -85,B 0,C 180,E1 17308.173,E2 17308.173} C_VEL
LIN {X 0,Y 308.858,Z 1012.173,A -85,B 0,C 180,E1 17311.994,E2 17311.994} C_VEL
LIN {X 0,Y 325.384,Z 999.835,A -85,B 0,C 180,E1 17314.341,E2 17314.341} C_VEL
LIN {X 0,Y 310.544,Z 1035.427,A -85,B 0,C 180,E1 17318.081,E2 17318.081} C_VEL
LIN {X 0,Y 294.384,Z 1066.86,A -85,B 0,C 180,E1 17322.865,E2 17322.865} C_VEL
LIN {X 0,Y 278.094,Z 1094.8,A -85,B 0,C 180,E1 17329.203,E2 17329.203} C_VEL
LIN {X 0,Y 264.331,Z 1116.816,A -85,B 0,C 180,E1 17336.641,E2 17336.641} C_VEL
LIN {X 0,Y 254.423,Z 1133.694,A -85,B 0,C 180,E1 17345.379,E2 17345.379} C_VEL
LIN {X 0,Y 249.092,Z 1144.344,A -85,B 0,C 180,E1 17354.123,E2 17354.123} C_VEL
LIN {X 0,Y 246.901,Z 1150.098,A -85,B 0,C 180,E1 17362.953,E2 17362.953} C_VEL
LIN {X 0,Y 246.862,Z 1151.497,A -85,B 0,C 180,E1 17369.998,E2 17369.998} C_VEL
LIN {X 0,Y 246.904,Z 1150.048,A -85,B 0,C 180,E1 17377.043,E2 17377.043} C_VEL
LIN {X 0,Y 249.129,Z 1144.256,A -85,B 0,C 180,E1 17385.871,E2 17385.871} C_VEL
LIN {X 0,Y 255.201,Z 1132.231,A -85,B 0,C 180,E1 17395.475,E2 17395.475} C_VEL
LIN {X 0,Y 265.844,Z 1114.419,A -85,B 0,C 180,E1 17404.212,E2 17404.212} C_VEL
LIN {X 0,Y 279.831,Z 1091.748,A -85,B 0,C 180,E1 17411.514,E2 17411.514} C_VEL
LIN {X 0,Y 295.572,Z 1064.568,A -85,B 0,C 180,E1 17417.423,E2 17417.423} C_VEL
LIN {X 0,Y 310.933,Z 1034.418,A -85,B 0,C 180,E1 17421.93,E2 17421.93} C_VEL
LIN {X 0,Y 325.239,Z 1000.598,A -85,B 0,C 180,E1 17425.428,E2 17425.428} C_VEL
LIN {X 0,Y 331.833,Z 981.012,A -85,B 0,C 180,E1 17427.002,E2 17427.002} C_VEL
LIN {X 0,Y 325.559,Z 958.392,A -85,B 0,C 180,E1 17432.693,E2 17432.693} C_VEL
LIN {X 0,Y 318.961,Z 941.077,A -85,B 0,C 180,E1 17438.418,E2 17438.418} C_VEL
LIN {X 0,Y 313.244,Z 928.921,A -85,B 0,C 180,E1 17444.17,E2 17444.17} C_VEL
LIN {X 0,Y 309.462,Z 920.246,A -85,B 0,C 180,E1 17450.03,E2 17450.03} C_VEL
LIN {X 0,Y 307.44,Z 916.604,A -85,B 0,C 180,E1 17458.59,E2 17458.59} C_VEL
LIN {X 0,Y 309.746,Z 921.368,A -85,B 0,C 180,E1 17466.491,E2 17466.491} C_VEL
LIN {X 0,Y 313.385,Z 929.8,A -85,B 0,C 180,E1 17471.971,E2 17471.971} C_VEL
LIN {X 0,Y 318.585,Z 941.206,A -85,B 0,C 180,E1 17477.28,E2 17477.28} C_VEL
LIN {X 0,Y 325.278,Z 959.816,A -85,B 0,C 180,E1 17483.306,E2 17483.306} C_VEL
LIN {X 0,Y 330.836,Z 981.615,A -85,B 0,C 180,E1 17488.636,E2 17488.636} C_VEL
LIN {X 0,Y 330.972,Z 985.379,A -85,B 0,C 180,E1 17489.303,E2 17489.303} C_VEL
LIN {X 0,Y 317.309,Z 1021.936,A -85,B 0,C 180,E1 17492.436,E2 17492.436} C_VEL
LIN {X 0,Y 302.032,Z 1055.914,A -85,B 0,C 180,E1 17496.671,E2 17496.671} C_VEL
LIN {X 0,Y 286.044,Z 1086.857,A -85,B 0,C 180,E1 17502.179,E2 17502.179} C_VEL
LIN {X 0,Y 271.071,Z 1113.892,A -85,B 0,C 180,E1 17509.116,E2 17509.116} C_VEL
LIN {X 0,Y 259.121,Z 1135.85,A -85,B 0,C 180,E1 17517.284,E2 17517.284} C_VEL
LIN {X 0,Y 251.448,Z 1151.879,A -85,B 0,C 180,E1 17526.019,E2 17526.019} C_VEL
LIN {X 0,Y 248.034,Z 1161.655,A -85,B 0,C 180,E1 17534.057,E2 17534.057} C_VEL
LIN {X 0,Y 246.638,Z 1167.902,A -85,B 0,C 180,E1 17542.949,E2 17542.949} C_VEL
LIN {X 0,Y 246.852,Z 1169.451,A -85,B 0,C 180,E1 17550.002,E2 17550.002} C_VEL
LIN {X 0,Y 246.636,Z 1167.908,A -85,B 0,C 180,E1 17557.054,E2 17557.054} C_VEL
LIN {X 0,Y 248.031,Z 1161.665,A -85,B 0,C 180,E1 17565.946,E2 17565.946} C_VEL
LIN {X 0,Y 252.025,Z 1150.5,A -85,B 0,C 180,E1 17574.871,E2 17574.871} C_VEL
LIN {X 0,Y 260.096,Z 1133.932,A -85,B 0,C 180,E1 17583.577,E2 17583.577} C_VEL
LIN {X 0,Y 272.774,Z 1110.988,A -85,B 0,C 180,E1 17591.769,E2 17591.769} C_VEL
LIN {X 0,Y 288.029,Z 1083.282,A -85,B 0,C 180,E1 17598.582,E2 17598.582} C_VEL
LIN {X 0,Y 304.198,Z 1051.557,A -85,B 0,C 180,E1 17603.985,E2 17603.985} C_VEL
LIN {X 0,Y 313.227,Z 1031.086,A -85,B 0,C 180,E1 17606.678,E2 17606.678} C_VEL
LIN {X 0,Y 290.151,Z 1042.317,A -85,B 0,C 180,E1 17610.352,E2 17610.352} C_VEL
LIN {X 0,Y 279.285,Z 1046.487,A -85,B 0,C 180,E1 17612.681,E2 17612.681} C_VEL
LIN {X 0,Y 270.823,Z 1051.617,A -85,B 0,C 180,E1 17614.064,E2 17614.064} C_VEL
LIN {X 0,Y 263.422,Z 1056.028,A -85,B 0,C 180,E1 17615.294,E2 17615.294} C_VEL
LIN {X 0,Y 262.553,Z 1056.314,A -85,B 0,C 180,E1 17615.544,E2 17615.544} C_VEL
LIN {X 0,Y 258.476,Z 1057.671,A -85,B 0,C 180,E1 17617.166,E2 17617.166} C_VEL
LIN {X 0,Y 251.587,Z 1068.467,A -85,B 0,C 180,E1 17623.39,E2 17623.39} C_VEL
LIN {X 0,Y 247.157,Z 1073.368,A -85,B 0,C 180,E1 17629.409,E2 17629.409} C_VEL
LIN {X 0,Y 244.202,Z 1073.437,A -85,B 0,C 180,E1 17636.444,E2 17636.444} C_VEL
LIN {X 0,Y 243.126,Z 1067.605,A -85,B 0,C 180,E1 17643.568,E2 17643.568} C_VEL
LIN {X 0,Y 243.565,Z 1057.413,A -85,B 0,C 180,E1 17649.84,E2 17649.84} C_VEL
LIN {X 0,Y 244.635,Z 1049.901,A -85,B 0,C 180,E1 17653.417,E2 17653.417} C_VEL
LIN {X 0,Y 261.99,Z 1042.637,A -85,B 0,C 180,E1 17662.373,E2 17662.373} C_VEL
LIN {X 0,Y 284.087,Z 1031.876,A -85,B 0,C 180,E1 17668.659,E2 17668.659} C_VEL
LIN {X 0,Y 306.787,Z 1018.494,A -85,B 0,C 180,E1 17672.875,E2 17672.875} C_VEL
LIN {X 0,Y 316.275,Z 1012.213,A -85,B 0,C 180,E1 17674.266,E2 17674.266} C_VEL
LIN {X 0,Y 299.867,Z 1047.537,A -85,B 0,C 180,E1 17678.494,E2 17678.494} C_VEL
LIN {X 0,Y 283.227,Z 1077.073,A -85,B 0,C 180,E1 17683.668,E2 17683.668} C_VEL
LIN {X 0,Y 267.307,Z 1102.415,A -85,B 0,C 180,E1 17690.256,E2 17690.256} C_VEL
LIN {X 0,Y 253.675,Z 1123.349,A -85,B 0,C 180,E1 17698.514,E2 17698.514} C_VEL
LIN {X 0,Y 244.958,Z 1137.743,A -85,B 0,C 180,E1 17707.272,E2 17707.272} C_VEL
LIN {X 0,Y 240.206,Z 1147.433,A -85,B 0,C 180,E1 17717.191,E2 17717.191} C_VEL
LIN {X 0,Y 238.83,Z 1151.442,A -85,B 0,C 180,E1 17726.363,E2 17726.363} C_VEL
LIN {X 0,Y 238.846,Z 1151.413,A -85,B 0,C 180,E1 17733.633,E2 17733.633} C_VEL
LIN {X 0,Y 240.224,Z 1147.351,A -85,B 0,C 180,E1 17742.828,E2 17742.828} C_VEL
LIN {X 0,Y 244.979,Z 1137.615,A -85,B 0,C 180,E1 17752.722,E2 17752.722} C_VEL
LIN {X 0,Y 254.899,Z 1121.417,A -85,B 0,C 180,E1 17762.316,E2 17762.316} C_VEL
LIN {X 0,Y 268.518,Z 1100.453,A -85,B 0,C 180,E1 17770.235,E2 17770.235} C_VEL
LIN {X 0,Y 284.729,Z 1074.408,A -85,B 0,C 180,E1 17776.761,E2 17776.761} C_VEL
LIN {X 0,Y 301.085,Z 1044.819,A -85,B 0,C 180,E1 17781.79,E2 17781.79} C_VEL
LIN {X 0,Y 316.486,Z 1011.847,A -85,B 0,C 180,E1 17785.614,E2 17785.614} C_VEL
LIN {X 0,Y 326.503,Z 985.655,A -85,B 0,C 180,E1 17787.788,E2 17787.788} C_VEL
LIN {X 0,Y 322.342,Z 967.244,A -85,B 0,C 180,E1 17792.427,E2 17792.427} C_VEL
LIN {X 0,Y 316.372,Z 949.361,A -85,B 0,C 180,E1 17798.233,E2 17798.233} C_VEL
LIN {X 0,Y 309.865,Z 933.608,A -85,B 0,C 180,E1 17805.771,E2 17805.771} C_VEL
LIN {X 0,Y 306.854,Z 927.435,A -85,B 0,C 180,E1 17811.118,E2 17811.118} C_VEL
LIN {X 0,Y 305.597,Z 924.282,A -85,B 0,C 180,E1 17818.582,E2 17818.582} C_VEL
LIN {X 0,Y 307.506,Z 928.878,A -85,B 0,C 180,E1 17826.234,E2 17826.234} C_VEL
LIN {X 0,Y 311.219,Z 937.908,A -85,B 0,C 180,E1 17832.156,E2 17832.156} C_VEL
LIN {X 0,Y 315.878,Z 949.558,A -85,B 0,C 180,E1 17837.433,E2 17837.433} C_VEL
LIN {X 0,Y 321.971,Z 968.66,A -85,B 0,C 180,E1 17843.559,E2 17843.559} C_VEL
LIN {X 0,Y 326.016,Z 987.494,A -85,B 0,C 180,E1 17848.216,E2 17848.216} C_VEL
LIN {X 0,Y 311.802,Z 1024.297,A -85,B 0,C 180,E1 17851.48,E2 17851.48} C_VEL
LIN {X 0,Y 295.632,Z 1058.586,A -85,B 0,C 180,E1 17855.875,E2 17855.875} C_VEL
LIN {X 0,Y 279.608,Z 1088.145,A -85,B 0,C 180,E1 17861.294,E2 17861.294} C_VEL
LIN {X 0,Y 264.665,Z 1113.876,A -85,B 0,C 180,E1 17868.044,E2 17868.044} C_VEL
LIN {X 0,Y 252.186,Z 1135.535,A -85,B 0,C 180,E1 17876.265,E2 17876.265} C_VEL
LIN {X 0,Y 243.435,Z 1152.854,A -85,B 0,C 180,E1 17886.155,E2 17886.155} C_VEL
LIN {X 0,Y 239.766,Z 1163.013,A -85,B 0,C 180,E1 17895.37,E2 17895.37} C_VEL
LIN {X 0,Y 238.762,Z 1167.612,A -85,B 0,C 180,E1 17902.715,E2 17902.715} C_VEL
LIN {X 0,Y 238.958,Z 1169.164,A -85,B 0,C 180,E1 17910.002,E2 17910.002} C_VEL
LIN {X 0,Y 238.76,Z 1167.619,A -85,B 0,C 180,E1 17917.288,E2 17917.288} C_VEL
LIN {X 0,Y 240.251,Z 1161.369,A -85,B 0,C 180,E1 17926.477,E2 17926.477} C_VEL
LIN {X 0,Y 244.597,Z 1150.193,A -85,B 0,C 180,E1 17935.68,E2 17935.68} C_VEL
LIN {X 0,Y 253.237,Z 1133.612,A -85,B 0,C 180,E1 17944.614,E2 17944.614} C_VEL
LIN {X 0,Y 266.633,Z 1110.651,A -85,B 0,C 180,E1 17952.959,E2 17952.959} C_VEL
LIN {X 0,Y 282.856,Z 1082.516,A -85,B 0,C 180,E1 17959.917,E2 17959.917} C_VEL
LIN {X 0,Y 299.75,Z 1050.48,A -85,B 0,C 180,E1 17965.349,E2 17965.349} C_VEL
LIN {X 0,Y 304.537,Z 1040.743,A -85,B 0,C 180,E1 17966.635,E2 17966.635} C_VEL
LIN {X 0,Y 280.216,Z 1050.89,A -85,B 0,C 180,E1 17970.904,E2 17970.904} C_VEL
LIN {X 0,Y 262.553,Z 1056.314,A -85,B 0,C 180,E1 17975.544,E2 17975.544} C_VEL
LIN {X 0,Y 254.595,Z 1060.464,A -85,B 0,C 180,E1 17977.302,E2 17977.302} C_VEL
LIN {X 0,Y 248.297,Z 1065.81,A -85,B 0,C 180,E1 17979.216,E2 17979.216} C_VEL
LIN {X 0,Y 242.005,Z 1073.38,A -85,B 0,C 180,E1 17985.507,E2 17985.507} C_VEL
LIN {X 0,Y 237.748,Z 1075.837,A -85,B 0,C 180,E1 17992.681,E2 17992.681} C_VEL
LIN {X 0,Y 235.669,Z 1072.49,A -85,B 0,C 180,E1 17999.998,E2 17999.998} C_VEL
LIN {X 0,Y 235.487,Z 1063.182,A -85,B 0,C 180,E1 18007.386,E2 18007.386} C_VEL
LIN {X 0,Y 235.924,Z 1057.323,A -85,B 0,C 180,E1 18010.63,E2 18010.63} C_VEL
LIN {X 0,Y 249.254,Z 1052.044,A -85,B 0,C 180,E1 18019.514,E2 18019.514} C_VEL
LIN {X 0,Y 271.873,Z 1042.369,A -85,B 0,C 180,E1 18027.348,E2 18027.348} C_VEL
LIN {X 0,Y 296.298,Z 1029.677,A -85,B 0,C 180,E1 18032.444,E2 18032.444} C_VEL
LIN {X 0,Y 306.695,Z 1023.378,A -85,B 0,C 180,E1 18034.045,E2 18034.045} C_VEL
LIN {X 0,Y 301.602,Z 1034.951,A -85,B 0,C 180,E1 18035.531,E2 18035.531} C_VEL
LIN {X 0,Y 284.25,Z 1066.683,A -85,B 0,C 180,E1 18040.334,E2 18040.334} C_VEL
LIN {X 0,Y 266.998,Z 1094.136,A -85,B 0,C 180,E1 18046.557,E2 18046.557} C_VEL
LIN {X 0,Y 251.525,Z 1116.716,A -85,B 0,C 180,E1 18054.301,E2 18054.301} C_VEL
LIN {X 0,Y 240.506,Z 1133.238,A -85,B 0,C 180,E1 18063.022,E2 18063.022} C_VEL
LIN {X 0,Y 233.718,Z 1144.927,A -85,B 0,C 180,E1 18073.049,E2 18073.049} C_VEL
LIN {X 0,Y 231.157,Z 1150.675,A -85,B 0,C 180,E1 18082.471,E2 18082.471} C_VEL
LIN {X 0,Y 231.09,Z 1152.07,A -85,B 0,C 180,E1 18089.998,E2 18089.998} C_VEL
LIN {X 0,Y 231.161,Z 1150.627,A -85,B 0,C 180,E1 18097.526,E2 18097.526} C_VEL
LIN {X 0,Y 233.746,Z 1144.841,A -85,B 0,C 180,E1 18106.946,E2 18106.946} C_VEL
LIN {X 0,Y 240.586,Z 1133.052,A -85,B 0,C 180,E1 18116.991,E2 18116.991} C_VEL
LIN {X 0,Y 252.448,Z 1115.372,A -85,B 0,C 180,E1 18126.141,E2 18126.141} C_VEL
LIN {X 0,Y 268.008,Z 1092.415,A -85,B 0,C 180,E1 18133.792,E2 18133.792} C_VEL
LIN {X 0,Y 284.55,Z 1066.047,A -85,B 0,C 180,E1 18139.664,E2 18139.664} C_VEL
LIN {X 0,Y 301.589,Z 1034.843,A -85,B 0,C 180,E1 18144.364,E2 18144.364} C_VEL
LIN {X 0,Y 317.181,Z 999.988,A -85,B 0,C 180,E1 18147.921,E2 18147.921} C_VEL
LIN {X 0,Y 321.374,Z 988.998,A -85,B 0,C 180,E1 18148.79,E2 18148.79} C_VEL
LIN {X 0,Y 317.193,Z 969.953,A -85,B 0,C 180,E1 18153.918,E2 18153.918} C_VEL
LIN {X 0,Y 312.216,Z 954.232,A -85,B 0,C 180,E1 18159.444,E2 18159.444} C_VEL
LIN {X 0,Y 307.399,Z 941.59,A -85,B 0,C 180,E1 18165.746,E2 18165.746} C_VEL
LIN {X 0,Y 304.692,Z 935.046,A -85,B 0,C 180,E1 18171.054,E2 18171.054} C_VEL
LIN {X 0,Y 303.433,Z 931.88,A -85,B 0,C 180,E1 18178.572,E2 18178.572} C_VEL
LIN {X 0,Y 305.161,Z 936.422,A -85,B 0,C 180,E1 18186.047,E2 18186.047} C_VEL
LIN {X 0,Y 308.647,Z 945.746,A -85,B 0,C 180,E1 18192.258,E2 18192.258} C_VEL
LIN {X 0,Y 313.546,Z 959.647,A -85,B 0,C 180,E1 18198.293,E2 18198.293} C_VEL
LIN {X 0,Y 318.877,Z 979.823,A -85,B 0,C 180,E1 18204.453,E2 18204.453} C_VEL
LIN {X 0,Y 320.591,Z 992.192,A -85,B 0,C 180,E1 18207.378,E2 18207.378} C_VEL
LIN {X 0,Y 304.472,Z 1030.818,A -85,B 0,C 180,E1 18210.928,E2 18210.928} C_VEL
LIN {X 0,Y 286.739,Z 1065.837,A -85,B 0,C 180,E1 18215.762,E2 18215.762} C_VEL
LIN {X 0,Y 269.446,Z 1095.881,A -85,B 0,C 180,E1 18221.88,E2 18221.88} C_VEL
LIN {X 0,Y 253.651,Z 1121.368,A -85,B 0,C 180,E1 18229.464,E2 18229.464} C_VEL
LIN {X 0,Y 241.816,Z 1141.481,A -85,B 0,C 180,E1 18238.364,E2 18238.364} C_VEL
LIN {X 0,Y 234.356,Z 1156.333,A -85,B 0,C 180,E1 18248.334,E2 18248.334} C_VEL
LIN {X 0,Y 231.261,Z 1165.404,A -85,B 0,C 180,E1 18258.674,E2 18258.674} C_VEL
LIN {X 0,Y 230.847,Z 1168.48,A -85,B 0,C 180,E1 18266.241,E2 18266.241} C_VEL
LIN {X 0,Y 231.055,Z 1168.876,A -85,B 0,C 180,E1 18270.002,E2 18270.002} C_VEL
LIN {X 0,Y 230.857,Z 1167.328,A -85,B 0,C 180,E1 18277.539,E2 18277.539} C_VEL
LIN {X 0,Y 232.508,Z 1161.073,A -85,B 0,C 180,E1 18287.042,E2 18287.042} C_VEL
LIN {X 0,Y 237.406,Z 1149.541,A -85,B 0,C 180,E1 18296.771,E2 18296.771} C_VEL
LIN {X 0,Y 247.124,Z 1132.286,A -85,B 0,C 180,E1 18306.14,E2 18306.14} C_VEL
LIN {X 0,Y 260.673,Z 1110.317,A -85,B 0,C 180,E1 18314.191,E2 18314.191} C_VEL
LIN {X 0,Y 276.76,Z 1083.68,A -85,B 0,C 180,E1 18320.909,E2 18320.909} C_VEL
LIN {X 0,Y 294.33,Z 1051.743,A -85,B 0,C 180,E1 18326.429,E2 18326.429} C_VEL
LIN {X 0,Y 295.366,Z 1049.547,A -85,B 0,C 180,E1 18326.747,E2 18326.747} C_VEL
LIN {X 0,Y 270.1,Z 1058.925,A -85,B 0,C 180,E1 18331.547,E2 18331.547} C_VEL
LIN {X 0,Y 249.678,Z 1063.811,A -85,B 0,C 180,E1 18338.08,E2 18338.08} C_VEL
LIN {X 0,Y 248.297,Z 1065.81,A -85,B 0,C 180,E1 18339.216,E2 18339.216} C_VEL
LIN {X 0,Y 240.731,Z 1072.093,A -85,B 0,C 180,E1 18342.633,E2 18342.633} C_VEL
LIN {X 0,Y 234.157,Z 1076.023,A -85,B 0,C 180,E1 18345.84,E2 18345.84} C_VEL
LIN {X 0,Y 233.693,Z 1076.349,A -85,B 0,C 180,E1 18346.356,E2 18346.356} C_VEL
LIN {X 0,Y 230.103,Z 1077.496,A -85,B 0,C 180,E1 18352.437,E2 18352.437} C_VEL
LIN {X 0,Y 227.877,Z 1073.696,A -85,B 0,C 180,E1 18359.998,E2 18359.998} C_VEL
LIN {X 0,Y 227.748,Z 1064.386,A -85,B 0,C 180,E1 18367.638,E2 18367.638} C_VEL
LIN {X 0,Y 241.028,Z 1059.145,A -85,B 0,C 180,E1 18378.302,E2 18378.302} C_VEL
LIN {X 0,Y 260.114,Z 1051.668,A -85,B 0,C 180,E1 18385.88,E2 18385.88} C_VEL
LIN {X 0,Y 282.961,Z 1041.358,A -85,B 0,C 180,E1 18391.444,E2 18391.444} C_VEL
LIN {X 0,Y 297.762,Z 1033.552,A -85,B 0,C 180,E1 18394.005,E2 18394.005} C_VEL
LIN {X 0,Y 280.374,Z 1064.964,A -85,B 0,C 180,E1 18398.713,E2 18398.713} C_VEL
LIN {X 0,Y 263.092,Z 1091.63,A -85,B 0,C 180,E1 18404.584,E2 18404.584} C_VEL
LIN {X 0,Y 246.803,Z 1114.514,A -85,B 0,C 180,E1 18412.155,E2 18412.155} C_VEL
LIN {X 0,Y 233.952,Z 1132.613,A -85,B 0,C 180,E1 18421.519,E2 18421.519} C_VEL
LIN {X 0,Y 227.007,Z 1143.454,A -85,B 0,C 180,E1 18430.517,E2 18430.517} C_VEL
LIN {X 0,Y 224.112,Z 1149.194,A -85,B 0,C 180,E1 18438.304,E2 18438.304} C_VEL
LIN {X 0,Y 223.038,Z 1152.018,A -85,B 0,C 180,E1 18446.106,E2 18446.106} C_VEL
LIN {X 0,Y 223.052,Z 1151.989,A -85,B 0,C 180,E1 18453.891,E2 18453.891} C_VEL
LIN {X 0,Y 224.639,Z 1147.985,A -85,B 0,C 180,E1 18463.643,E2 18463.643} C_VEL
LIN {X 0,Y 230.195,Z 1138.207,A -85,B 0,C 180,E1 18474.272,E2 18474.272} C_VEL
LIN {X 0,Y 241.385,Z 1122.036,A -85,B 0,C 180,E1 18484.368,E2 18484.368} C_VEL
LIN {X 0,Y 256.615,Z 1100.803,A -85,B 0,C 180,E1 18492.657,E2 18492.657} C_VEL
LIN {X 0,Y 274.428,Z 1074.428,A -85,B 0,C 180,E1 18499.341,E2 18499.341} C_VEL
LIN {X 0,Y 292.066,Z 1044.496,A -85,B 0,C 180,E1 18504.415,E2 18504.415} C_VEL
LIN {X 0,Y 308.687,Z 1010.821,A -85,B 0,C 180,E1 18508.229,E2 18508.229} C_VEL
LIN {X 0,Y 316.201,Z 991.743,A -85,B 0,C 180,E1 18509.955,E2 18509.955} C_VEL
LIN {X 0,Y 311.905,Z 971.644,A -85,B 0,C 180,E1 18515.836,E2 18515.836} C_VEL
LIN {X 0,Y 307.606,Z 957.504,A -85,B 0,C 180,E1 18521.363,E2 18521.363} C_VEL
LIN {X 0,Y 303.954,Z 947.481,A -85,B 0,C 180,E1 18527.049,E2 18527.049} C_VEL
LIN {X 0,Y 302.169,Z 942.438,A -85,B 0,C 180,E1 18531.357,E2 18531.357} C_VEL
LIN {X 0,Y 301.182,Z 939.557,A -85,B 0,C 180,E1 18537.12,E2 18537.12} C_VEL
LIN {X 0,Y 301.59,Z 941.574,A -85,B 0,C 180,E1 18542.879,E2 18542.879} C_VEL
LIN {X 0,Y 302.807,Z 945.07,A -85,B 0,C 180,E1 18546.686,E2 18546.686} C_VEL
LIN {X 0,Y 306.216,Z 954.694,A -85,B 0,C 180,E1 18552.856,E2 18552.856} C_VEL
LIN {X 0,Y 310.339,Z 967.999,A -85,B 0,C 180,E1 18558.489,E2 18558.489} C_VEL
LIN {X 0,Y 314.42,Z 986.391,A -85,B 0,C 180,E1 18564.159,E2 18564.159} C_VEL
LIN {X 0,Y 315.667,Z 994.407,A -85,B 0,C 180,E1 18566.226,E2 18566.226} C_VEL
LIN {X 0,Y 299.725,Z 1031.667,A -85,B 0,C 180,E1 18569.745,E2 18569.745} C_VEL
LIN {X 0,Y 281.811,Z 1065.81,A -85,B 0,C 180,E1 18574.468,E2 18574.468} C_VEL
LIN {X 0,Y 263.987,Z 1095.537,A -85,B 0,C 180,E1 18580.541,E2 18580.541} C_VEL
LIN {X 0,Y 247.347,Z 1121.164,A -85,B 0,C 180,E1 18588.265,E2 18588.265} C_VEL
LIN {X 0,Y 234.371,Z 1141.875,A -85,B 0,C 180,E1 18597.718,E2 18597.718} C_VEL
LIN {X 0,Y 226.429,Z 1156.806,A -85,B 0,C 180,E1 18608.316,E2 18608.316} C_VEL
LIN {X 0,Y 223.401,Z 1165.11,A -85,B 0,C 180,E1 18618.27,E2 18618.27} C_VEL
LIN {X 0,Y 222.952,Z 1168.192,A -85,B 0,C 180,E1 18626.108,E2 18626.108} C_VEL
LIN {X 0,Y 223.151,Z 1168.589,A -85,B 0,C 180,E1 18630.002,E2 18630.002} C_VEL
LIN {X 0,Y 222.967,Z 1167.038,A -85,B 0,C 180,E1 18637.808,E2 18637.808} C_VEL
LIN {X 0,Y 224.774,Z 1160.778,A -85,B 0,C 180,E1 18647.648,E2 18647.648} C_VEL
LIN {X 0,Y 229.9,Z 1149.582,A -85,B 0,C 180,E1 18657.455,E2 18657.455} C_VEL
LIN {X 0,Y 240.465,Z 1131.967,A -85,B 0,C 180,E1 18667.307,E2 18667.307} C_VEL
LIN {X 0,Y 254.778,Z 1109.983,A -85,B 0,C 180,E1 18675.494,E2 18675.494} C_VEL
LIN {X 0,Y 271.888,Z 1082.906,A -85,B 0,C 180,E1 18682.341,E2 18682.341} C_VEL
LIN {X 0,Y 285.938,Z 1058.547,A -85,B 0,C 180,E1 18686.707,E2 18686.707} C_VEL
LIN {X 0,Y 260.202,Z 1066.3,A -85,B 0,C 180,E1 18692.258,E2 18692.258} C_VEL
LIN {X 0,Y 240.769,Z 1069.968,A -85,B 0,C 180,E1 18699.285,E2 18699.285} C_VEL
LIN {X 0,Y 233.693,Z 1076.349,A -85,B 0,C 180,E1 18706.356,E2 18706.356} C_VEL
LIN {X 0,Y 229.231,Z 1078.06,A -85,B 0,C 180,E1 18709.374,E2 18709.374} C_VEL
LIN {X 0,Y 221.708,Z 1078.658,A -85,B 0,C 180,E1 18714.017,E2 18714.017} C_VEL
LIN {X 0,Y 221.415,Z 1078.292,A -85,B 0,C 180,E1 18714.577,E2 18714.577} C_VEL
LIN {X 0,Y 219.802,Z 1072.833,A -85,B 0,C 180,E1 18722.031,E2 18722.031} C_VEL
LIN {X 0,Y 219.867,Z 1071.398,A -85,B 0,C 180,E1 18723.946,E2 18723.946} C_VEL
LIN {X 0,Y 235.735,Z 1064.84,A -85,B 0,C 180,E1 18738.728,E2 18738.728} C_VEL
LIN {X 0,Y 255.148,Z 1057.786,A -85,B 0,C 180,E1 18746.423,E2 18746.423} C_VEL
LIN {X 0,Y 281.137,Z 1046.641,A -85,B 0,C 180,E1 18752.58,E2 18752.58} C_VEL
LIN {X 0,Y 288.026,Z 1043.161,A -85,B 0,C 180,E1 18753.775,E2 18753.775} C_VEL
LIN {X 0,Y 285.549,Z 1048.66,A -85,B 0,C 180,E1 18754.723,E2 18754.723} C_VEL
LIN {X 0,Y 266.883,Z 1078.453,A -85,B 0,C 180,E1 18760.01,E2 18760.01} C_VEL
LIN {X 0,Y 248.681,Z 1104.016,A -85,B 0,C 180,E1 18766.93,E2 18766.93} C_VEL
LIN {X 0,Y 233.304,Z 1124.253,A -85,B 0,C 180,E1 18775.396,E2 18775.396} C_VEL
LIN {X 0,Y 222.826,Z 1138.626,A -85,B 0,C 180,E1 18784.867,E2 18784.867} C_VEL
LIN {X 0,Y 216.883,Z 1148.341,A -85,B 0,C 180,E1 18795.855,E2 18795.855} C_VEL
LIN {X 0,Y 215.136,Z 1152.306,A -85,B 0,C 180,E1 18805.962,E2 18805.962} C_VEL
LIN {X 0,Y 215.15,Z 1152.278,A -85,B 0,C 180,E1 18814.034,E2 18814.034} C_VEL
LIN {X 0,Y 216.894,Z 1148.276,A -85,B 0,C 180,E1 18824.141,E2 18824.141} C_VEL
LIN {X 0,Y 222.858,Z 1138.503,A -85,B 0,C 180,E1 18835.126,E2 18835.126} C_VEL
LIN {X 0,Y 234.749,Z 1122.346,A -85,B 0,C 180,E1 18845.484,E2 18845.484} C_VEL
LIN {X 0,Y 250.702,Z 1101.227,A -85,B 0,C 180,E1 18853.868,E2 18853.868} C_VEL
LIN {X 0,Y 268.173,Z 1076.49,A -85,B 0,C 180,E1 18860.287,E2 18860.287} C_VEL
LIN {X 0,Y 286.878,Z 1046.03,A -85,B 0,C 180,E1 18865.554,E2 18865.554} C_VEL
LIN {X 0,Y 304.251,Z 1012.071,A -85,B 0,C 180,E1 18869.429,E2 18869.429} C_VEL
LIN {X 0,Y 311.077,Z 995.734,A -85,B 0,C 180,E1 18870.879,E2 18870.879} C_VEL
LIN {X 0,Y 307.516,Z 976.512,A -85,B 0,C 180,E1 18876.807,E2 18876.807} C_VEL
LIN {X 0,Y 303.623,Z 962.721,A -85,B 0,C 180,E1 18882.593,E2 18882.593} C_VEL
LIN {X 0,Y 300.583,Z 953.416,A -85,B 0,C 180,E1 18888.379,E2 18888.379} C_VEL
LIN {X 0,Y 299.63,Z 950.055,A -85,B 0,C 180,E1 18891.283,E2 18891.283} C_VEL
LIN {X 0,Y 298.646,Z 947.069,A -85,B 0,C 180,E1 18897.096,E2 18897.096} C_VEL
LIN {X 0,Y 299.051,Z 949.087,A -85,B 0,C 180,E1 18902.903,E2 18902.903} C_VEL
LIN {X 0,Y 301.033,Z 955.046,A -85,B 0,C 180,E1 18908.679,E2 18908.679} C_VEL
LIN {X 0,Y 304.592,Z 967.091,A -85,B 0,C 180,E1 18915.128,E2 18915.128} C_VEL
LIN {X 0,Y 308.333,Z 983.477,A -85,B 0,C 180,E1 18921.091,E2 18921.091} C_VEL
LIN {X 0,Y 310.289,Z 999.036,A -85,B 0,C 180,E1 18925.374,E2 18925.374} C_VEL
LIN {X 0,Y 294.396,Z 1033.888,A -85,B 0,C 180,E1 18928.678,E2 18928.678} C_VEL
LIN {X 0,Y 276.219,Z 1067.104,A -85,B 0,C 180,E1 18933.354,E2 18933.354} C_VEL
LIN {X 0,Y 257.662,Z 1096.693,A -85,B 0,C 180,E1 18939.533,E2 18939.533} C_VEL
LIN {X 0,Y 240.431,Z 1121.967,A -85,B 0,C 180,E1 18947.393,E2 18947.393} C_VEL
LIN {X 0,Y 227.416,Z 1141.565,A -85,B 0,C 180,E1 18956.605,E2 18956.605} C_VEL
LIN {X 0,Y 218.802,Z 1156.611,A -85,B 0,C 180,E1 18967.631,E2 18967.631} C_VEL
LIN {X 0,Y 215.568,Z 1164.817,A -85,B 0,C 180,E1 18977.838,E2 18977.838} C_VEL
LIN {X 0,Y 215.035,Z 1167.903,A -85,B 0,C 180,E1 18985.964,E2 18985.964} C_VEL
LIN {X 0,Y 215.247,Z 1168.302,A -85,B 0,C 180,E1 18990.002,E2 18990.002} C_VEL
LIN {X 0,Y 215.167,Z 1165.931,A -85,B 0,C 180,E1 18999.906,E2 18999.906} C_VEL
LIN {X 0,Y 217.066,Z 1160.482,A -85,B 0,C 180,E1 19008.296,E2 19008.296} C_VEL
LIN {X 0,Y 222.632,Z 1149.278,A -85,B 0,C 180,E1 19018.431,E2 19018.431} C_VEL
LIN {X 0,Y 232.99,Z 1133.112,A -85,B 0,C 180,E1 19027.866,E2 19027.866} C_VEL
LIN {X 0,Y 248.013,Z 1111.202,A -85,B 0,C 180,E1 19036.383,E2 19036.383} C_VEL
LIN {X 0,Y 266.258,Z 1083.66,A -85,B 0,C 180,E1 19043.512,E2 19043.512} C_VEL
LIN {X 0,Y 276.974,Z 1065.983,A -85,B 0,C 180,E1 19046.864,E2 19046.864} C_VEL
LIN {X 0,Y 249.74,Z 1073.322,A -85,B 0,C 180,E1 19053.251,E2 19053.251} C_VEL
LIN {X 0,Y 231.416,Z 1075.866,A -85,B 0,C 180,E1 19060.905,E2 19060.905} C_VEL
LIN {X 0,Y 224.598,Z 1079.161,A -85,B 0,C 180,E1 19068.331,E2 19068.331} C_VEL
LIN {X 0,Y 221.415,Z 1078.292,A -85,B 0,C 180,E1 19074.577,E2 19074.577} C_VEL
LIN {X 0,Y 216.808,Z 1077.58,A -85,B 0,C 180,E1 19078.994,E2 19078.994} C_VEL
LIN {X 0,Y 213.891,Z 1076.916,A -85,B 0,C 180,E1 19083.567,E2 19083.567} C_VEL
LIN {X 0,Y 230.383,Z 1070.489,A -85,B 0,C 180,E1 19099.18,E2 19099.18} C_VEL
LIN {X 0,Y 250.024,Z 1063.683,A -85,B 0,C 180,E1 19107.008,E2 19107.008} C_VEL
LIN {X 0,Y 276.365,Z 1053.032,A -85,B 0,C 180,E1 19113.215,E2 19113.215} C_VEL
LIN {X 0,Y 278.498,Z 1052.115,A -85,B 0,C 180,E1 19113.615,E2 19113.615} C_VEL
LIN {X 0,Y 277.47,Z 1055.01,A -85,B 0,C 180,E1 19114.302,E2 19114.302} C_VEL
LIN {X 0,Y 258.437,Z 1083.479,A -85,B 0,C 180,E1 19119.736,E2 19119.736} C_VEL
LIN {X 0,Y 240.301,Z 1107.511,A -85,B 0,C 180,E1 19126.744,E2 19126.744} C_VEL
LIN {X 0,Y 225.347,Z 1126.229,A -85,B 0,C 180,E1 19135.169,E2 19135.169} C_VEL
LIN {X 0,Y 214.736,Z 1140.015,A -85,B 0,C 180,E1 19144.969,E2 19144.969} C_VEL
LIN {X 0,Y 209.136,Z 1148.631,A -85,B 0,C 180,E1 19155.319,E2 19155.319} C_VEL
LIN {X 0,Y 207.25,Z 1152.594,A -85,B 0,C 180,E1 19165.808,E2 19165.808} C_VEL
LIN {X 0,Y 207.263,Z 1152.566,A -85,B 0,C 180,E1 19174.187,E2 19174.187} C_VEL
LIN {X 0,Y 209.148,Z 1148.567,A -85,B 0,C 180,E1 19184.676,E2 19184.676} C_VEL
LIN {X 0,Y 215.587,Z 1138.799,A -85,B 0,C 180,E1 19196.035,E2 19196.035} C_VEL
LIN {X 0,Y 228.213,Z 1122.654,A -85,B 0,C 180,E1 19206.662,E2 19206.662} C_VEL
LIN {X 0,Y 244.698,Z 1101.9,A -85,B 0,C 180,E1 19215.065,E2 19215.065} C_VEL
LIN {X 0,Y 263.112,Z 1076.842,A -85,B 0,C 180,E1 19221.633,E2 19221.633} C_VEL
LIN {X 0,Y 282.467,Z 1046.427,A -85,B 0,C 180,E1 19226.881,E2 19226.881} C_VEL
LIN {X 0,Y 300.77,Z 1011.514,A -85,B 0,C 180,E1 19230.824,E2 19230.824} C_VEL
LIN {X 0,Y 305.991,Z 999.395,A -85,B 0,C 180,E1 19231.929,E2 19231.929} C_VEL
LIN {X 0,Y 302.964,Z 980.803,A -85,B 0,C 180,E1 19237.991,E2 19237.991} C_VEL
LIN {X 0,Y 299.409,Z 966.617,A -85,B 0,C 180,E1 19244.498,E2 19244.498} C_VEL
LIN {X 0,Y 296.83,Z 957.602,A -85,B 0,C 180,E1 19251.2,E2 19251.2} C_VEL
LIN {X 0,Y 295.992,Z 954.559,A -85,B 0,C 180,E1 19257.07,E2 19257.07} C_VEL
LIN {X 0,Y 296.318,Z 956.508,A -85,B 0,C 180,E1 19262.93,E2 19262.93} C_VEL
LIN {X 0,Y 298.062,Z 962.753,A -85,B 0,C 180,E1 19268.766,E2 19268.766} C_VEL
LIN {X 0,Y 301.138,Z 974.853,A -85,B 0,C 180,E1 19275.214,E2 19275.214} C_VEL
LIN {X 0,Y 304.382,Z 991.98,A -85,B 0,C 180,E1 19281.378,E2 19281.378} C_VEL
LIN {X 0,Y 305.423,Z 1001.45,A -85,B 0,C 180,E1 19284.14,E2 19284.14} C_VEL
LIN {X 0,Y 288.468,Z 1037.543,A -85,B 0,C 180,E1 19287.756,E2 19287.756} C_VEL
LIN {X 0,Y 269.457,Z 1070.474,A -85,B 0,C 180,E1 19292.557,E2 19292.557} C_VEL
LIN {X 0,Y 250.595,Z 1099.084,A -85,B 0,C 180,E1 19298.808,E2 19298.808} C_VEL
LIN {X 0,Y 233.582,Z 1122.77,A -85,B 0,C 180,E1 19306.472,E2 19306.472} C_VEL
LIN {X 0,Y 220.528,Z 1141.329,A -85,B 0,C 180,E1 19315.471,E2 19315.471} C_VEL
LIN {X 0,Y 211.253,Z 1156.311,A -85,B 0,C 180,E1 19326.786,E2 19326.786} C_VEL
LIN {X 0,Y 207.724,Z 1164.523,A -85,B 0,C 180,E1 19337.371,E2 19337.371} C_VEL
LIN {X 0,Y 207.143,Z 1167.615,A -85,B 0,C 180,E1 19345.81,E2 19345.81} C_VEL
LIN {X 0,Y 207.359,Z 1168.015,A -85,B 0,C 180,E1 19350.002,E2 19350.002} C_VEL
LIN {X 0,Y 207.186,Z 1166.457,A -85,B 0,C 180,E1 19358.407,E2 19358.407} C_VEL
LIN {X 0,Y 209.256,Z 1160.499,A -85,B 0,C 180,E1 19368.594,E2 19368.594} C_VEL
LIN {X 0,Y 215.437,Z 1148.973,A -85,B 0,C 180,E1 19379.473,E2 19379.473} C_VEL
LIN {X 0,Y 226.337,Z 1133.08,A -85,B 0,C 180,E1 19389.015,E2 19389.015} C_VEL
LIN {X 0,Y 242.636,Z 1110.549,A -85,B 0,C 180,E1 19397.89,E2 19397.89} C_VEL
LIN {X 0,Y 261.346,Z 1083.482,A -85,B 0,C 180,E1 19404.922,E2 19404.922} C_VEL
LIN {X 0,Y 267.608,Z 1073.196,A -85,B 0,C 180,E1 19407.065,E2 19407.065} C_VEL
LIN {X 0,Y 250.072,Z 1077.658,A -85,B 0,C 180,E1 19411.03,E2 19411.03} C_VEL
LIN {X 0,Y 232.634,Z 1080.665,A -85,B 0,C 180,E1 19417.014,E2 19417.014} C_VEL
LIN {X 0,Y 217.803,Z 1080.944,A -85,B 0,C 180,E1 19426.942,E2 19426.942} C_VEL
LIN {X 0,Y 213.694,Z 1079.759,A -85,B 0,C 180,E1 19434.428,E2 19434.428} C_VEL
LIN {X 0,Y 213.891,Z 1076.916,A -85,B 0,C 180,E1 19443.567,E2 19443.567} C_VEL
LIN {X 0,Y 213.563,Z 1078.144,A -85,B 0,C 180,E1 19448.25,E2 19448.25} C_VEL
LIN {X 0,Y 214.806,Z 1079.24,A -85,B 0,C 180,E1 19452.903,E2 19452.903} C_VEL
LIN {X 0,Y 235.737,Z 1072.523,A -85,B 0,C 180,E1 19464.58,E2 19464.58} C_VEL
LIN {X 0,Y 263.676,Z 1062.546,A -85,B 0,C 180,E1 19472.38,E2 19472.38} C_VEL
LIN {X 0,Y 269.171,Z 1060.346,A -85,B 0,C 180,E1 19473.467,E2 19473.467} C_VEL
LIN {X 0,Y 267.768,Z 1063.402,A -85,B 0,C 180,E1 19474.218,E2 19474.218} C_VEL
LIN {X 0,Y 248.907,Z 1089.693,A -85,B 0,C 180,E1 19479.791,E2 19479.791} C_VEL
LIN {X 0,Y 230.784,Z 1112.339,A -85,B 0,C 180,E1 19487.139,E2 19487.139} C_VEL
LIN {X 0,Y 216.059,Z 1129.776,A -85,B 0,C 180,E1 19495.898,E2 19495.898} C_VEL
LIN {X 0,Y 205.435,Z 1143.035,A -85,B 0,C 180,E1 19506.758,E2 19506.758} C_VEL
LIN {X 0,Y 200.744,Z 1150.064,A -85,B 0,C 180,E1 19516.92,E2 19516.92} C_VEL
LIN {X 0,Y 199.35,Z 1152.882,A -85,B 0,C 180,E1 19525.642,E2 19525.642} C_VEL
LIN {X 0,Y 199.362,Z 1152.854,A -85,B 0,C 180,E1 19534.354,E2 19534.354} C_VEL
LIN {X 0,Y 201.424,Z 1148.858,A -85,B 0,C 180,E1 19545.252,E2 19545.252} C_VEL
LIN {X 0,Y 208.389,Z 1139.093,A -85,B 0,C 180,E1 19557.006,E2 19557.006} C_VEL
LIN {X 0,Y 221.797,Z 1122.962,A -85,B 0,C 180,E1 19567.906,E2 19567.906} C_VEL
LIN {X 0,Y 239.531,Z 1101.618,A -85,B 0,C 180,E1 19576.626,E2 19576.626} C_VEL
LIN {X 0,Y 259.4,Z 1075.475,A -85,B 0,C 180,E1 19583.376,E2 19583.376} C_VEL
LIN {X 0,Y 278.821,Z 1045.695,A -85,B 0,C 180,E1 19588.417,E2 19588.417} C_VEL
LIN {X 0,Y 297.025,Z 1011.923,A -85,B 0,C 180,E1 19592.166,E2 19592.166} C_VEL
LIN {X 0,Y 300.926,Z 1002.903,A -85,B 0,C 180,E1 19593.079,E2 19593.079} C_VEL
LIN {X 0,Y 298.472,Z 985.094,A -85,B 0,C 180,E1 19599.204,E2 19599.204} C_VEL
LIN {X 0,Y 295.728,Z 972.945,A -85,B 0,C 180,E1 19605.17,E2 19605.17} C_VEL
LIN {X 0,Y 293.921,Z 965.161,A -85,B 0,C 180,E1 19611.112,E2 19611.112} C_VEL
LIN {X 0,Y 293.117,Z 961.953,A -85,B 0,C 180,E1 19617.041,E2 19617.041} C_VEL
LIN {X 0,Y 293.437,Z 963.913,A -85,B 0,C 180,E1 19622.959,E2 19622.959} C_VEL
LIN {X 0,Y 295.09,Z 971.581,A -85,B 0,C 180,E1 19629.6,E2 19629.6} C_VEL
LIN {X 0,Y 297.529,Z 982.818,A -85,B 0,C 180,E1 19635.404,E2 19635.404} C_VEL
LIN {X 0,Y 299.894,Z 999.491,A -85,B 0,C 180,E1 19641.396,E2 19641.396} C_VEL
LIN {X 0,Y 300.132,Z 1006.201,A -85,B 0,C 180,E1 19643.248,E2 19643.248} C_VEL
LIN {X 0,Y 281.837,Z 1042.515,A -85,B 0,C 180,E1 19646.957,E2 19646.957} C_VEL
LIN {X 0,Y 261.424,Z 1075.823,A -85,B 0,C 180,E1 19652.109,E2 19652.109} C_VEL
LIN {X 0,Y 241.275,Z 1104.45,A -85,B 0,C 180,E1 19658.866,E2 19658.866} C_VEL
LIN {X 0,Y 223.623,Z 1127.944,A -85,B 0,C 180,E1 19667.386,E2 19667.386} C_VEL
LIN {X 0,Y 210.377,Z 1145.836,A -85,B 0,C 180,E1 19677.333,E2 19677.333} C_VEL
LIN {X 0,Y 202.217,Z 1159.02,A -85,B 0,C 180,E1 19689.139,E2 19689.139} C_VEL
LIN {X 0,Y 199.899,Z 1164.229,A -85,B 0,C 180,E1 19696.868,E2 19696.868} C_VEL
LIN {X 0,Y 199.224,Z 1167.326,A -85,B 0,C 180,E1 19705.643,E2 19705.643} C_VEL
LIN {X 0,Y 199.454,Z 1167.727,A -85,B 0,C 180,E1 19710.002,E2 19710.002} C_VEL
LIN {X 0,Y 199.308,Z 1166.032,A -85,B 0,C 180,E1 19719.065,E2 19719.065} C_VEL
LIN {X 0,Y 201.524,Z 1160.321,A -85,B 0,C 180,E1 19729.173,E2 19729.173} C_VEL
LIN {X 0,Y 208.324,Z 1148.671,A -85,B 0,C 180,E1 19740.584,E2 19740.584} C_VEL
LIN {X 0,Y 221.252,Z 1131.071,A -85,B 0,C 180,E1 19751.173,E2 19751.173} C_VEL
LIN {X 0,Y 237.986,Z 1108.987,A -85,B 0,C 180,E1 19759.774,E2 19759.774} C_VEL
LIN {X 0,Y 257.117,Z 1082.485,A -85,B 0,C 180,E1 19766.559,E2 19766.559} C_VEL
LIN {X 0,Y 257.862,Z 1080.207,A -85,B 0,C 180,E1 19767.259,E2 19767.259} C_VEL
LIN {X 0,Y 235.406,Z 1084.856,A -85,B 0,C 180,E1 19773.243,E2 19773.243} C_VEL
LIN {X 0,Y 220.34,Z 1086.396,A -85,B 0,C 180,E1 19779.905,E2 19779.905} C_VEL
LIN {X 0,Y 208.319,Z 1085.238,A -85,B 0,C 180,E1 19791.641,E2 19791.641} C_VEL
LIN {X 0,Y 214.806,Z 1079.24,A -85,B 0,C 180,E1 19812.903,E2 19812.903} C_VEL
LIN {X 0,Y 217.792,Z 1079.97,A -85,B 0,C 180,E1 19817.458,E2 19817.458} C_VEL
LIN {X 0,Y 222.45,Z 1080.308,A -85,B 0,C 180,E1 19821.809,E2 19821.809} C_VEL
LIN {X 0,Y 247.73,Z 1072.293,A -85,B 0,C 180,E1 19830.545,E2 19830.545} C_VEL
LIN {X 0,Y 259.815,Z 1068.092,A -85,B 0,C 180,E1 19833.319,E2 19833.319} C_VEL
LIN {X 0,Y 257.733,Z 1071.723,A -85,B 0,C 180,E1 19834.229,E2 19834.229} C_VEL
LIN {X 0,Y 237.163,Z 1098.313,A -85,B 0,C 180,E1 19840.697,E2 19840.697} C_VEL
LIN {X 0,Y 219.253,Z 1119.023,A -85,B 0,C 180,E1 19848.537,E2 19848.537} C_VEL
LIN {X 0,Y 204.379,Z 1135.767,A -85,B 0,C 180,E1 19858.76,E2 19858.76} C_VEL
LIN {X 0,Y 195.696,Z 1146.381,A -85,B 0,C 180,E1 19869.622,E2 19869.622} C_VEL
LIN {X 0,Y 191.869,Z 1152.119,A -85,B 0,C 180,E1 19880.917,E2 19880.917} C_VEL
LIN {X 0,Y 191.611,Z 1153.506,A -85,B 0,C 180,E1 19889.998,E2 19889.998} C_VEL
LIN {X 0,Y 191.895,Z 1152.073,A -85,B 0,C 180,E1 19899.078,E2 19899.078} C_VEL
LIN {X 0,Y 195.721,Z 1146.302,A -85,B 0,C 180,E1 19910.371,E2 19910.371} C_VEL
LIN {X 0,Y 205.998,Z 1133.902,A -85,B 0,C 180,E1 19922.576,E2 19922.576} C_VEL
LIN {X 0,Y 222.359,Z 1115.53,A -85,B 0,C 180,E1 19932.915,E2 19932.915} C_VEL
LIN {X 0,Y 241.283,Z 1093.125,A -85,B 0,C 180,E1 19940.706,E2 19940.706} C_VEL
LIN {X 0,Y 262.033,Z 1065.454,A -85,B 0,C 180,E1 19946.829,E2 19946.829} C_VEL
LIN {X 0,Y 281.709,Z 1034.434,A -85,B 0,C 180,E1 19951.271,E2 19951.271} C_VEL
LIN {X 0,Y 295.548,Z 1007.899,A -85,B 0,C 180,E1 19953.928,E2 19953.928} C_VEL
LIN {X 0,Y 294.771,Z 995.23,A -85,B 0,C 180,E1 19958.14,E2 19958.14} C_VEL
LIN {X 0,Y 292.818,Z 983.321,A -85,B 0,C 180,E1 19963.481,E2 19963.481} C_VEL
LIN {X 0,Y 291.038,Z 974.619,A -85,B 0,C 180,E1 19969.218,E2 19969.218} C_VEL
LIN {X 0,Y 290.082,Z 970.699,A -85,B 0,C 180,E1 19974.01,E2 19974.01} C_VEL
LIN {X 0,Y 290.066,Z 969.275,A -85,B 0,C 180,E1 19977.01,E2 19977.01} C_VEL
LIN {X 0,Y 290.286,Z 971.231,A -85,B 0,C 180,E1 19982.991,E2 19982.991} C_VEL
LIN {X 0,Y 291.723,Z 978.897,A -85,B 0,C 180,E1 19989.552,E2 19989.552} C_VEL
LIN {X 0,Y 293.794,Z 990.896,A -85,B 0,C 180,E1 19995.698,E2 19995.698} C_VEL
LIN {X 0,Y 295.367,Z 1008.684,A -85,B 0,C 180,E1 20001.963,E2 20001.963} C_VEL
LIN {X 0,Y 277.399,Z 1043.489,A -85,B 0,C 180,E1 20005.632,E2 20005.632} C_VEL
LIN {X 0,Y 257.144,Z 1075.463,A -85,B 0,C 180,E1 20010.556,E2 20010.556} C_VEL
LIN {X 0,Y 236.21,Z 1104.122,A -85,B 0,C 180,E1 20017.316,E2 20017.316} C_VEL
LIN {X 0,Y 217.485,Z 1127.623,A -85,B 0,C 180,E1 20025.88,E2 20025.88} C_VEL
LIN {X 0,Y 203.405,Z 1145.609,A -85,B 0,C 180,E1 20036.136,E2 20036.136} C_VEL
LIN {X 0,Y 195.159,Z 1157.746,A -85,B 0,C 180,E1 20047.177,E2 20047.177} C_VEL
LIN {X 0,Y 192.076,Z 1163.936,A -85,B 0,C 180,E1 20056.323,E2 20056.323} C_VEL
LIN {X 0,Y 191.308,Z 1167.036,A -85,B 0,C 180,E1 20065.463,E2 20065.463} C_VEL
LIN {X 0,Y 191.566,Z 1167.44,A -85,B 0,C 180,E1 20070.002,E2 20070.002} C_VEL
LIN {X 0,Y 191.434,Z 1165.877,A -85,B 0,C 180,E1 20079.104,E2 20079.104} C_VEL
LIN {X 0,Y 194.136,Z 1159.535,A -85,B 0,C 180,E1 20090.636,E2 20090.636} C_VEL
LIN {X 0,Y 201.274,Z 1148.366,A -85,B 0,C 180,E1 20101.778,E2 20101.778} C_VEL
LIN {X 0,Y 215.087,Z 1130.759,A -85,B 0,C 180,E1 20112.626,E2 20112.626} C_VEL
LIN {X 0,Y 232.727,Z 1108.659,A -85,B 0,C 180,E1 20121.33,E2 20121.33} C_VEL
LIN {X 0,Y 248.73,Z 1087.544,A -85,B 0,C 180,E1 20126.949,E2 20126.949} C_VEL
LIN {X 0,Y 248.897,Z 1086.583,A -85,B 0,C 180,E1 20127.341,E2 20127.341} C_VEL
LIN {X 0,Y 229.993,Z 1090.027,A -85,B 0,C 180,E1 20132.561,E2 20132.561} C_VEL
LIN {X 0,Y 209.07,Z 1091.558,A -85,B 0,C 180,E1 20143.161,E2 20143.161} C_VEL
LIN {X 0,Y 200.922,Z 1088.396,A -85,B 0,C 180,E1 20159.998,E2 20159.998} C_VEL
LIN {X 0,Y 212.968,Z 1083.184,A -85,B 0,C 180,E1 20176.518,E2 20176.518} C_VEL
LIN {X 0,Y 222.45,Z 1080.308,A -85,B 0,C 180,E1 20181.809,E2 20181.809} C_VEL
LIN {X 0,Y 235.544,Z 1079.997,A -85,B 0,C 180,E1 20189.347,E2 20189.347} C_VEL
LIN {X 0,Y 236.875,Z 1079.634,A -85,B 0,C 180,E1 20189.754,E2 20189.754} C_VEL
LIN {X 0,Y 249.892,Z 1075.418,A -85,B 0,C 180,E1 20193.04,E2 20193.04} C_VEL
LIN {X 0,Y 247.972,Z 1079.119,A -85,B 0,C 180,E1 20194.153,E2 20194.153} C_VEL
LIN {X 0,Y 226.503,Z 1104.929,A -85,B 0,C 180,E1 20201.23,E2 20201.23} C_VEL
LIN {X 0,Y 207.402,Z 1125.517,A -85,B 0,C 180,E1 20210.35,E2 20210.35} C_VEL
LIN {X 0,Y 194.119,Z 1139.798,A -85,B 0,C 180,E1 20220.821,E2 20220.821} C_VEL
LIN {X 0,Y 186.025,Z 1149.501,A -85,B 0,C 180,E1 20233.446,E2 20233.446} C_VEL
LIN {X 0,Y 183.551,Z 1153.458,A -85,B 0,C 180,E1 20245.266,E2 20245.266} C_VEL
LIN {X 0,Y 183.707,Z 1153.793,A -85,B 0,C 180,E1 20249.998,E2 20249.998} C_VEL
LIN {X 0,Y 184.075,Z 1152.362,A -85,B 0,C 180,E1 20259.467,E2 20259.467} C_VEL
LIN {X 0,Y 188.214,Z 1146.617,A -85,B 0,C 180,E1 20271.183,E2 20271.183} C_VEL
LIN {X 0,Y 198.711,Z 1134.772,A -85,B 0,C 180,E1 20283.4,E2 20283.4} C_VEL
LIN {X 0,Y 215.568,Z 1116.895,A -85,B 0,C 180,E1 20293.914,E2 20293.914} C_VEL
LIN {X 0,Y 235.794,Z 1094.045,A -85,B 0,C 180,E1 20302.054,E2 20302.054} C_VEL
LIN {X 0,Y 256.688,Z 1067.325,A -85,B 0,C 180,E1 20308.055,E2 20308.055} C_VEL
LIN {X 0,Y 276.908,Z 1036.721,A -85,B 0,C 180,E1 20312.497,E2 20312.497} C_VEL
LIN {X 0,Y 290.354,Z 1012.053,A -85,B 0,C 180,E1 20315.015,E2 20315.015} C_VEL
LIN {X 0,Y 290.626,Z 1005.146,A -85,B 0,C 180,E1 20317.146,E2 20317.146} C_VEL
LIN {X 0,Y 289.329,Z 992.339,A -85,B 0,C 180,E1 20322.56,E2 20322.56} C_VEL
LIN {X 0,Y 287.558,Z 981.695,A -85,B 0,C 180,E1 20329.383,E2 20329.383} C_VEL
LIN {X 0,Y 286.883,Z 977.974,A -85,B 0,C 180,E1 20333.943,E2 20333.943} C_VEL
LIN {X 0,Y 286.858,Z 976.538,A -85,B 0,C 180,E1 20336.976,E2 20336.976} C_VEL
LIN {X 0,Y 287.054,Z 978.53,A -85,B 0,C 180,E1 20343.025,E2 20343.025} C_VEL
LIN {X 0,Y 288.072,Z 986.347,A -85,B 0,C 180,E1 20349.674,E2 20349.674} C_VEL
LIN {X 0,Y 289.482,Z 996.926,A -85,B 0,C 180,E1 20355.16,E2 20355.16} C_VEL
LIN {X 0,Y 290.401,Z 1012.663,A -85,B 0,C 180,E1 20360.935,E2 20360.935} C_VEL
LIN {X 0,Y 271.762,Z 1046.695,A -85,B 0,C 180,E1 20364.555,E2 20364.555} C_VEL
LIN {X 0,Y 251.053,Z 1077.859,A -85,B 0,C 180,E1 20369.489,E2 20369.489} C_VEL
LIN {X 0,Y 230.409,Z 1104.871,A -85,B 0,C 180,E1 20376.016,E2 20376.016} C_VEL
LIN {X 0,Y 211.582,Z 1127.307,A -85,B 0,C 180,E1 20384.308,E2 20384.308} C_VEL
LIN {X 0,Y 196.436,Z 1145.482,A -85,B 0,C 180,E1 20394.933,E2 20394.933} C_VEL
LIN {X 0,Y 187.641,Z 1157.445,A -85,B 0,C 180,E1 20406.207,E2 20406.207} C_VEL
LIN {X 0,Y 184.282,Z 1163.642,A -85,B 0,C 180,E1 20415.732,E2 20415.732} C_VEL
LIN {X 0,Y 183.389,Z 1166.747,A -85,B 0,C 180,E1 20425.266,E2 20425.266} C_VEL
LIN {X 0,Y 183.658,Z 1167.153,A -85,B 0,C 180,E1 20430.002,E2 20430.002} C_VEL
LIN {X 0,Y 183.565,Z 1165.587,A -85,B 0,C 180,E1 20439.498,E2 20439.498} C_VEL
LIN {X 0,Y 186.526,Z 1159.239,A -85,B 0,C 180,E1 20451.519,E2 20451.519} C_VEL
LIN {X 0,Y 195.377,Z 1146.792,A -85,B 0,C 180,E1 20464.067,E2 20464.067} C_VEL
LIN {X 0,Y 210.397,Z 1128.826,A -85,B 0,C 180,E1 20474.967,E2 20474.967} C_VEL
LIN {X 0,Y 229.168,Z 1106.491,A -85,B 0,C 180,E1 20483.516,E2 20483.516} C_VEL
LIN {X 0,Y 239.799,Z 1092.655,A -85,B 0,C 180,E1 20487.458,E2 20487.458} C_VEL
LIN {X 0,Y 216.002,Z 1095.976,A -85,B 0,C 180,E1 20495.13,E2 20495.13} C_VEL
LIN {X 0,Y 203.104,Z 1096.4,A -85,B 0,C 180,E1 20502.651,E2 20502.651} C_VEL
LIN {X 0,Y 196.071,Z 1092.154,A -85,B 0,C 180,E1 20524.426,E2 20524.426} C_VEL
LIN {X 0,Y 213.522,Z 1086.381,A -85,B 0,C 180,E1 20540.762,E2 20540.762} C_VEL
LIN {X 0,Y 236.875,Z 1079.634,A -85,B 0,C 180,E1 20549.754,E2 20549.754} C_VEL
LIN {X 0,Y 239.437,Z 1080.448,A -85,B 0,C 180,E1 20551.401,E2 20551.401} C_VEL
LIN {X 0,Y 237.941,Z 1085.682,A -85,B 0,C 180,E1 20553.796,E2 20553.796} C_VEL
LIN {X 0,Y 235.19,Z 1089.54,A -85,B 0,C 180,E1 20554.966,E2 20554.966} C_VEL
LIN {X 0,Y 214.648,Z 1112.234,A -85,B 0,C 180,E1 20562.279,E2 20562.279} C_VEL
LIN {X 0,Y 196.436,Z 1130.665,A -85,B 0,C 180,E1 20571.926,E2 20571.926} C_VEL
LIN {X 0,Y 184.004,Z 1143.372,A -85,B 0,C 180,E1 20583.088,E2 20583.088} C_VEL
LIN {X 0,Y 177.506,Z 1150.934,A -85,B 0,C 180,E1 20595.171,E2 20595.171} C_VEL
LIN {X 0,Y 175.678,Z 1153.745,A -85,B 0,C 180,E1 20605.053,E2 20605.053} C_VEL
LIN {X 0,Y 175.803,Z 1154.081,A -85,B 0,C 180,E1 20609.998,E2 20609.998} C_VEL
LIN {X 0,Y 176.233,Z 1152.652,A -85,B 0,C 180,E1 20619.892,E2 20619.892} C_VEL
LIN {X 0,Y 180.472,Z 1147.206,A -85,B 0,C 180,E1 20631.62,E2 20631.62} C_VEL
LIN {X 0,Y 190.816,Z 1136.224,A -85,B 0,C 180,E1 20643.739,E2 20643.739} C_VEL
LIN {X 0,Y 206.937,Z 1120.098,A -85,B 0,C 180,E1 20654.033,E2 20654.033} C_VEL
LIN {X 0,Y 227.1,Z 1098.692,A -85,B 0,C 180,E1 20662.345,E2 20662.345} C_VEL
LIN {X 0,Y 249.197,Z 1072.08,A -85,B 0,C 180,E1 20668.764,E2 20668.764} C_VEL
LIN {X 0,Y 270.114,Z 1042.181,A -85,B 0,C 180,E1 20673.362,E2 20673.362} C_VEL
LIN {X 0,Y 285.997,Z 1014.607,A -85,B 0,C 180,E1 20676.308,E2 20676.308} C_VEL
LIN {X 0,Y 285.27,Z 1000.169,A -85,B 0,C 180,E1 20682.234,E2 20682.234} C_VEL
LIN {X 0,Y 284.26,Z 990.974,A -85,B 0,C 180,E1 20687.701,E2 20687.701} C_VEL
LIN {X 0,Y 283.373,Z 985.116,A -85,B 0,C 180,E1 20693.868,E2 20693.868} C_VEL
LIN {X 0,Y 283.409,Z 983.694,A -85,B 0,C 180,E1 20696.939,E2 20696.939} C_VEL
LIN {X 0,Y 283.42,Z 983.955,A -85,B 0,C 180,E1 20700.001,E2 20700.001} C_VEL
LIN {X 0,Y 283.764,Z 988.712,A -85,B 0,C 180,E1 20706.127,E2 20706.127} C_VEL
LIN {X 0,Y 284.748,Z 998.043,A -85,B 0,C 180,E1 20712.28,E2 20712.28} C_VEL
LIN {X 0,Y 285.428,Z 1011.786,A -85,B 0,C 180,E1 20718.158,E2 20718.158} C_VEL
LIN {X 0,Y 285.149,Z 1017.211,A -85,B 0,C 180,E1 20719.876,E2 20719.876} C_VEL
LIN {X 0,Y 264.711,Z 1052.384,A -85,B 0,C 180,E1 20723.771,E2 20723.771} C_VEL
